FUNCTION_BLOCK FB_CapPreScrewer
VAR_INPUT
	bEnable								: BOOL;		//Zezwolenie na pracę
	bEstop								: BOOL;		//Stop awaryjny nieaktywny
	bHoming								: BOOL;		//Zezwolenie na wykonanie bazowania
	bIgnoreError						: BOOL;		//Ignorowania błędów cyklu pracy
	
	bReset								: BOOL;		//Reset błędu, jeśli w stanie "eError
	bManualMovement						: BOOL;		//Zezwolenie na ruchy ręcznę
	
	bRun								: BOOL;		//Rozkaz uruchomienia zakręcarki
	bPreRun								: BOOL;		//Przygotowanie stacji do pracy
	bSimulationEna						: BOOL;		//Tryb symulacji
	bPlacePermission					: BOOL;		//Zezwolenenie na wkładanie nakrentki w butelkę
	bMover1InPlacePos					: BOOL;		//Wózek 1 na pozycji Place
	bMover2InPlacePos					: BOOL;		//Wózek 2 na pozycji Place

	bCapSuckerVacumOk1					: BOOL;		//Sygnał podciśnienia na ssawce nakrętki 1
	bCapSuckerVacumOk2					: BOOL;		//Sygnał podciśnienia na ssawce nakrętki 2
	bCapSuckerVacumOk3					: BOOL;		//Sygnał podciśnienia na ssawce nakrętki 3
	bCapSuckerVacumOk4					: BOOL;		//Sygnał podciśnienia na ssawce nakrętki 4
	
	bStrawCatcherOut					: BOOL;		//Sygnał z krańcówki - wysunięty łapacz słomek
	bStrawCatcherIn						: BOOL;		//Sygnał z krańcówki - wysunięty łapacz słomek
	
	bStrawCatcherOpen1					: BOOL;		//Sygnał z krańcówki - otwart łapacz słomek 1
	bStrawCatcherOpen2					: BOOL;		//Sygnał z krańcówki - otwart łapacz słomek 2
	bStrawCatcherOpen3					: BOOL;		//Sygnał z krańcówki - otwart łapacz słomek 3
	bStrawCatcherOpen4					: BOOL;		//Sygnał z krańcówki - otwart łapacz słomek 4
	bSetEncoderOffsetAxisZ				: BOOL;		//Ustaw pozycję enkodera osi Z 
	
	stCommandsIn						: ST_CapPreScrewerCommandsIn;		

	stParameters						: ST_CapPreScrewerParameters;
	stMoverStatus						: ST_MoverState;
	
	iStationIndex						: UDINT;		//Numer stacji 
	wsStationName						: WSTRING;	//Nazwa stacji
	
END_VAR

VAR_OUTPUT
	eState							: E_Station;			//Stan ogólny bloku
	eRunningState					: E_CapPreScrewer; 		//Stan załapywarki
	bHomingDone						: BOOL;					//Stacja zbazowana
	bError							: BOOL;						//Błąd stacji
	udiErrorID						: UDINT;					//Nr błędu zakręcarki
	sErrorDescription				: STRING(200);				//Opis błędu
	sErrorDescription2				: STRING(200);				//Opis błędu
	sErrorStationName				: STRING;					//Nazwa stacj
	
	udiCartesianXServoErrorNr		: UDINT;					//Nr błędu serwa poziomego X
	udiCartesianZServoErrorNr		: UDINT;					//Nr błędu serwa pionowego Y
	udiPreScrewerServoErrorNr		: UDINT;					//Nr błędu serwa obrotowego załapywarki
	udiCatcherServoErrorNr			: UDINT;					//Nr błędu serwo pionowego uchwytu słomek
	
	_OUTPUT_						: BOOL;
	bBottleGrippers					: BOOL;						//Sygnał do zaworu - łapania szyjek butelek

	bCapSucker 						: ARRAY [1..4] OF BOOL;		//Sygnał do zaworu - zassij nakrętkę
	//bCapSucker2						: BOOL;						//Sygnał do zaworu - zassij nakrętkę 2
	//bCapSucker3						: BOOL;						//Sygnał do zaworu - zassij nakrętkę 3
	//bCapSucker4						: BOOL;						//Sygnał do zaworu - zassij nakrętkę 4
	
	bCapBlower1						: BOOL;						//Sygnał do zaworu - wydmuchaj nakrętkę 1
	bCapBlower2						: BOOL;						//Sygnał do zaworu - wydmuchaj nakrętkę 2
	bCapBlower3						: BOOL;						//Sygnał do zaworu - wydmuchaj nakrętkę 3
	bCapBlower4						: BOOL;						//Sygnał do zaworu - wydmuchaj nakrętkę 4
	
	bCapCatcher1					: BOOL;						//Sygnał do zaworu - złap nakrętkę 1
	bCapCatcher2					: BOOL;						//Sygnał do zaworu - złap nakrętkę 2
	bCapCatcher3					: BOOL;						//Sygnał do zaworu - złap nakrętkę 3
	bCapCatcher4					: BOOL;						//Sygnał do zaworu - złap nakrętkę 4
	
	bStrawCatchersOpen				: BOOL;						//Sygnał do zaworu - otwórz chwytaki słomek
	bStrawCatchersClose				: BOOL;						//Sygnał do zaworu - zamknij chwytaki słomek
	
	bStrawCatcherActuatorOut		: BOOL;						//Sygnał do zaworu - wysuń łapacz słomek
	bStrawCatcherActuatorIn			: BOOL;						//Sygnał do zaworu - wsuń łapacz słomek
	bMissingCaps					: BOOL;						//Żadna nakretka nie zostala pobrana
	
	bCycleDone						: BOOL;						//Cykl zakończono
	bCycleNotDone					: BOOL;						//Nie zakończono cyklu przestawiania wózków
	aCapPresence					: ARRAY [1..4] OF BOOL;		//jakie nakretki zostaly odlozone do butelek
	bAxisYSafePos					: BOOL;						//Bezpieczna pozycja osi Y dla przejazdu mówerów
	bCartesianSafePos				: BOOL;						//Bezpieczna pozycja kartezjana dla przejazdu mówerów
	bRejectDone						: BOOL;						// Zakończony odrzut
END_VAR

VAR_IN_OUT
	bStepButton						: BOOL; 		//Następny krok sekwencji	

	bManualBottleGripperUp			: BOOL;			//Ręczny ruch Jisang
	bManualBottleGripperDown		: BOOL;			//Ręczny ruch Jisang
	
	bManualCartesianYJogPlus		: BOOL;			//Ruch ręczny podajnika zamknięć 
	bManualCartesianYJogMinus		: BOOL;			//Ruch ręczny podajnika zamknięć 
	bManualCartesianZJogPlus		: BOOL;			//Ruch ręczny podajnika zamknięć 
	bManualCartesianZJogMinus		: BOOL;			//Ruch ręczny podajnika zamknięć 
	
	bManualPreScrewerJogPlus		: BOOL;
	bManualPreScrewerJogMinus		: BOOL;
	
	bManualCatcherJogPlus			: BOOL;
	bManualCatcherJogMinus			: BOOL;

	bManualCapSucker1				: BOOL;						//Ręczne sterowanie zaworu - zassij nakrętkę 1
	bmanualCapSucker2				: BOOL;						//Ręczne sterowanie - zassij nakrętkę 2
	bManualCapSucker3				: BOOL;						//Ręczne sterowanie - zassij nakrętkę 3
	bManualCapSucker4				: BOOL;						//Ręczne sterowanie - zassij nakrętkę 4
	                                
	bManualCapBlower1				: BOOL;						//Ręczne sterowanie - wydmuchaj nakrętkę 1
	bManualCapBlower2				: BOOL;						//Ręczne sterowanie - wydmuchaj nakrętkę 2
	bManualCapBlower3				: BOOL;						//Ręczne sterowanie - wydmuchaj nakrętkę 3
	bManualCapBlower4				: BOOL;						//Ręczne sterowanie - wydmuchaj nakrętkę 4
	
	bManualCapCatcher1				: BOOL;						//Ręczne sterowanie - złap nakrętkę 1
	bManualCapCatcher2				: BOOL;						//Ręczne sterowanie - złap nakrętkę 2
	bManualCapCatcher3				: BOOL;						//Ręczne sterowanie - złap nakrętkę 3
	bManualCapCatcher4				: BOOL;						//Ręczne sterowanie - złap nakrętkę 4
	
	bManualStrawCatchersOpen		: BOOL;						//Ręczne sterowanie - zamknij chwytaki słomek
	bManualStrawCatchersClose		: BOOL;                     //Ręczne sterowanie - otwórz chwytaki słomek
	                                  
	bManualStrawCatcherActuatorOut	: BOOL;						//Ręczne sterowanie - wysuń łapacz słomek
	bManualStrawCatcherActuatorIn	: BOOL;                     //Ręczne sterowanie - wsuń łapacz słomek
	
	CartesianYAxisRef				: AXIS_REF;		//Struktura sterowania NC dla serwa przesuwania poziomego
	CartesianZAxisRef				: AXIS_REF;		//Struktura sterowania NC dla serwa przesuwania pionowego
	PreScrewerAxisRef				: AXIS_REF;		//Struktura sterowania NC dla serwa załapywania nakrętek
	CatcherAxisRef					: AXIS_REF;		//Struktura sterowania NC dla serwa prowadzenia słomki
	bAdvancedHoming: BOOL;
END_VAR

VAR
	fbStrawCatcherLift				: FB_Checker;

	diMover1VacuumRetry				: ARRAY [1..4] OF DINT;					// Ilość prób pobrania wózek 1, słoty 1..4
	diMover2VacuumRetry				: ARRAY [1..4] OF DINT;					// Ilość prób pobrania wózek 2, słoty 1..4
	
	tonDelayServoOn					: TON;
	
	mcCartesianYManualMove			: MC_JOG; 			// Blok ruchu ręcznego 
	mcCartesianZManualMove			: MC_JOG; 			// Blok ruchu ręcznego
	mcPreScrewerManualMove			: MC_JOG; 			// Blok ruchu ręcznego
	mcCatcherManualMove				: MC_JOG; 			// Blok ruchu ręcznego
	
	mcCartesianYStop				: MC_Stop;			// Trwałe zatrzymywanie Serwo
	mcCartesianZStop				: MC_Stop;			// Trwałe zatrzymywanie Serwo
	mcPreScrewerStop				: MC_Stop;			// Trwałe zatrzymywanie Serwo
	mcCatcherStop					: MC_Stop;			// Trwałe zatrzymywanie Serwo
	
	mcCatcherHalt				: MC_Halt;			// Trwałe zatrzymywanie Serwo
	
//	mcMover1MoveVelocity		: MC_MoveVelocity;		// Ruch prędkościowy
//	mcMover2MoveVelocity		: MC_MoveVelocity;		// Ruch prędkościowy
//	mcMover1MoveVelocity2		: MC_MoveVelocity;		// Ruch prędkościowy
//	mcMover2MoveVelocity2		: MC_MoveVelocity;		// Ruch prędkościowy	
//	mcMover1MoveRelative		: MC_MoveRelative; 		// Ruch relatywny
	
	mcCartesianYMoveAbsolute	: MC_MoveAbsolute; 		// Ruch absolutny
	mcCartesianYMoveRelative	: MC_MoveRelative;		// Ruch względny
	mcCartesianZMoveAbsolute	: MC_MoveAbsolute; 		// Ruch absolutny
	mcCartesianZMoveAbsolute2	: MC_MoveAbsolute; 		// Ruch absolutny
	mcPreScrewerMoveAbsolute	: MC_MoveAbsolute; 		// Ruch absolutny
	mcPreScrewerMoveRelative	: MC_MoveRelative; 		// Ruch względny
	mcCatcherMoveAbsolute		: MC_MoveAbsolute; 		// Ruch absolutny
	
	fbAxisYPositioningOffset	: FB_CoEAX8000SetPositionOffset;
	fbAxisZPositioningOffset	: FB_CoEAX8000SetPositionOffset;
	
	mcCartesianYPower			: MC_Power;			 	// Zasilanie napędu
	mcCartesianZPower			: MC_Power;			 	// Zasilanie napędu
	mcPreScrewerPower			: MC_Power;			 	// Zasilanie napędu
	mcCatcherPower				: MC_Power;			 	// Zasilanie napędu
	
	mcPreScrewerHome			: MC_Home;	
	
	bCartesianYServoPower		: BOOL;					// Zmienna sterujaca zasilaniem serwo
	bCartesianZServoPower		: BOOL;					// Zmienna sterujaca zasilaniem serwo	
	bPreScrewerPower			: BOOL;					// Zmienna sterujaca zasilaniem serwo
	bCatcherPower				: BOOL;					// Zmienna sterujaca zasilaniem serwo
	
	fbCartesianYHardReset		: FB_SoEReset; 			// Blok twardego resetu serwa
	fbCartesianZHardReset		: FB_SoEReset; 			// Blok twardego resetu serwa
	fbPreScrewerHardReset		: FB_SoEReset; 			// Blok twardego resetu serwa
	fbCatcherHardReset			: FB_SoEReset; 			// Blok twardego resetu serwa
	mcCartesianYSoftReset		: MC_Reset; 			// blok łagodnego resetu serwa 
	mcCartesianZSoftReset		: MC_Reset; 			// blok łagodnego resetu serwa
	mcPreScrewerSoftReset		: MC_Reset; 			// blok łagodnego resetu serwa
	mcCatcherSoftReset			: MC_Reset; 			// blok łagodnego resetu serwa
	
	(*Bledy, Resetowanie*)
	tonResetting						: TON;
	rtResetCommands						: R_TRIG;
	tonActualMotor1TemperatureTooHigh	: TON;
	tonActualMotor2TemperatureTooHigh	: TON;
		
	bStateError							: BOOL;
	
	eLastState					: E_Station;			// Stan ogólny bloku
	eLastRunningState			: E_CapPreScrewer;		// Stan podbloku
	eLastStateTemp				: E_Station;			// Stan ogólny bloku
	//eLastRunningStateTemp		: E_CapFeeder;		// Stan podbloku
	
	(*Casy od różnych stanów*)
	iAbortingCASE				: INT;
	iStoppingCase 				: INT;
	iHomingCase					: INT;
	iErrorResseting2			: INT;
	iTestResetting				: INT;
	iCountAborting				: INT;
	
	(*Filtry czujników*)
	tonSuckedOk					: ARRAY [1..4] OF TON;
	//tonSuckedOk2				: TON;
	//tonSuckedOk3				: TON;
	//tonSuckedOk4				: TON;
	
	tonStrawCatcherIn			: TON;
	tonStrawCatcherOut			: TON;
	
	tonStrawCatcher1Open		: TON;
	tonStrawCatcher2Open		: TON;
	tonStrawCatcher3Open		: TON;
	tonStrawCatcher4Open		: TON;
	
	tonStrawCatcher1Close		: TON;
	tonStrawCatcher2Close		: TON;
	tonStrawCatcher3Close		: TON;
	tonStrawCatcher4Close		: TON;
	
	//Czasówki do obsługi błędów siłowników
	tonErrorStrawCatcherIn		: TON;
	tonErrorStrawCatcherOut		: TON;
	
	tonErrorStrawCatcherOpen1	: TON;
	tonErrorStrawCatcherOpen2	: TON;
	tonErrorStrawCatcherOpen3	: TON;
	tonErrorStrawCatcherOpen4	: TON;
	
	//Czasówki do obsługi problemu z zasysaniem
	tonErrorSuckerVacum1		: TON;
	tonErrorSuckerVacum2		: TON;
	tonErrorSuckerVacum3		: TON;
	tonErrorSuckerVacum4		: TON;
	tonCapCatcher				: TON;
	
	tonBlowOFF					: TON;
	bCapsBlowON					: BOOL;
	
	tonVacuumWatchdog			: TON;
	i: INT;
	
	tonBlowerON				: ARRAY [1..4] OF TON;	//Cap blowing timers
		
	tonPlacePermission			: TON;
	rtPlacePermission			: R_TRIG;
	bGripperOpen: BOOL;
	bStopAllowed: BOOL;
	
//	fbBottleCatch									: fb
	eBottleCatch1State								:E_Station; 						// Stan chwytaka stabilizujšcego pod podajnikiem nakrętek
	eBottleCatch2State								:E_Station; 						// Stan chwytaka stabilizujšcego pod podajnikiem nakrętek
	eBottleCatch3State								:E_Station; 						// Stan chwytaka stabilizujšcego pod podajnikiem nakrętek
	eBottleCatch4State								:E_Station; 						// Stan chwytaka stabilizujšcego pod podajnikiem nakrętek
	eBottleCatch1RunningState						:E_CatchStationState; 				// Poprzedni stan chwytaka pod podajnikiem nakrętek
	eBottleCatch2RunningState						:E_CatchStationState; 				// Poprzedni stan chwytaka pod podajnikiem nakrętek
	eBottleCatch3RunningState						:E_CatchStationState; 				// Poprzedni stan chwytaka pod podajnikiem nakrętek
	eBottleCatch4RunningState						:E_CatchStationState; 				// Poprzedni stan chwytaka pod podajnikiem nakręte
	fbBottleCatch1State								:FB_State;
	fbBottleCatch2State								:FB_State;
	fbBottleCatch3State								:FB_State;
	fbBottleCatch4State								:FB_State;
	
	IbBottleCatchHeightMotorEncoderPulse			: BOOL;									// Sygnał impulsów enkodera siłownika	
                                            
                                                    
    QbBottleCatchHeightUpCmd              			: BOOL;  								// Zmienna sterownika bezpośrednio sterująca siłownikiem w górę 
    QbBottleCatchHeightDownCmd            			: BOOL;									// Zmienna sterownika bezpośrednio sterująca siłownikiem w dół 	
	bBottleCatcherCatchTemp							: BOOL;
	rtRun											: R_TRIG;
	bTestStrawCatcher								: BOOL;
	bTestError										: BOOL;
	bCatcHActuator1									: BOOL;
	bCatcHActuator2									: BOOL;
	bCatcHActuator3									: BOOL;
	bCatcHActuator4									: BOOL;
                                                	
	bCollisionWithMoverArea							: BOOL;
	bCollisionError									: BOOL;
	bCollision1Error								: BOOL;
	bCollision2Error								: BOOL;
	rtCollisionError								: R_TRIG;
	tonCollisionError								: TON;
	bCapBlow1										: BOOL;
	bCapBlow2										: BOOL;
	bCapBlow3										: BOOL;
	bCapBlow4										: BOOL;
	bPlaceDone										: BOOL;
	bTestCatch										: BOOL;
	iDisablingCase									: INT;
	bAdditionalBlow									: BOOL;
	bAxisYInPosition								: BOOL;
	bAxisZInPosition								: BOOL;
	bAxisZInPosition1								: BOOL;
	bAxisZInPosition2								: BOOL;
	bHomingWithoutJiesang							: BOOL;
	bCapLost										: ARRAY [1..4] OF BOOL;
	bAnyCapLost										: BOOL;

	trStepButton: R_TRIG;
	diManualModeCase								: DINT;
	bAxisYInHomePos									: BOOL;
	bAxisZInHomePos									: BOOL;
	bAxisZInTopPos									: BOOL;
	bAxisStrawCatcherHomePos						: BOOL;
	bCartesianInHomePos								: BOOL;										//Kartezjan znajduje sie na poz. home
	bCartesianInTopPos								: BOOL;
	bCartesianReady									: BOOL;										//Kartezjan gotowy do sekwencji
	rtCheckVacuumPart4								: R_TRIG;	


	FB_AxisY_ADS_Read								: FB_EcCoESdoRead;
	uiAxisY_ADS_Read								: UINT;
	tonAxisY_ADS_Read							    : TON;
	
	stAxisY_ADS										: ST_ADS_Read_Write;
	iAxisY_ADS_ReadCase								: INT;
	
	ftAxisY_ADS_Read								: F_TRIG;
	
	ftAxisY_ADS_Write								: F_TRIG;
	
	bSetPosition									: BOOL;
	FB_AxisY_ADS_Write								: FB_EcCoESdoWrite;
	tonAxisYLagDetction								: TON;		
	bCartesianInReadyPos							: BOOL;
	lrPreScrewerAxisSavedPosition					: LREAL;
	lrAxisZSavedPosition							: LREAL;
	
	bChangeSpeedRightLeft							: BOOL;
	rtPendantRightLeftFast							: R_TRIG;
	ftPendantRightLeftFast							: F_TRIG;
	bChangeSpeedUpDown								: BOOL;
	rtPendantUpDownFast								: R_TRIG;
	ftPendantUpDownFast								: F_TRIG;
	
	bAnyCapPresence									: BOOL;		//Obecna przynajmniej jedna nasadka
	tonWaitInPlacePos								: TON;
	diPreSCrewerHomePos								: DINT;

	//Synchronizacja osi podczas prowadzenia slomki
	fbGearInAxisZ									: MC_GearInDyn;
	fbGearInAxisZ_Screwer							: MC_GearIn;	
	fbGearInCatcherAxis								: MC_GearInDyn;
	fbGearOutAxisZ									: MC_GearOut;
	fbGearOutCatcherAxis							: MC_GearOut;
	fbVirtualAxis									: FB_AxisAX8000;
	fbGearInPos										: MC_GearInPos; 
	VirtualEna										: BOOL := TRUE;
	
	fbCamTableSelectAxisZ							: MC_CamTableSelect;
	fbCamInAxisZ									: MC_CamIn;
	fbCamOutAxisZ									: MC_CamOut;
	fbCamTableSelectCatcher							: MC_CamTableSelect;
	fbCamInAxisCatcher								: MC_CamIn;
	fbCamOutAxisCatcher								: MC_CamOut;	
	
	stCamTableIdAxisZ								: MC_CAM_ID;
	stCamTableAxisZRef								: MC_CAM_REF;
	arrTableAxisZ									: ARRAY[0..2, 0..1] OF LREAL;
	stCamTableIdCatcher								: MC_CAM_ID;
	stCamTableCatcherRef							: MC_CAM_REF;
	arrTableCatcher									: ARRAY[0..2, 0..1] OF LREAL;
	
	nAxisYSafetyState			AT%I*				: BYTE;	//Satatus safety 
	nAxisZSafetyState			AT%I*				: BYTE;	//Satatus safety 
	nAxisScrewSafetyState		AT%I*				: BYTE;	//Satatus safety 
	nAxisCatcherSafetyState		AT%I*				: BYTE;	//Satatus safety 
	
	uiAxisYTorqueLimit			AT%Q*				: UINT;
	
	rtChoseRecipe									: R_TRIG;
	tonCapCatcher1Open								: TON;
	bVirtualMove									: BOOL;		//Absolutny ruch  wirtualnej osi
	rtMove											: R_TRIG;
	ftMove											: F_TRIG;
	bVirtualAxisMove1								: BOOL;		//Ruch 1 wirtualnej osi
	bVirtualAxisMove2								: BOOL;		//Ruch 2 wirtualnej osi
	
	nMoveId											: INT;		//
	stVirtualMove_Out								: Tc2_MC2.ST_McOutputs;
	stVirtualMove1_Out								: Tc2_MC2.ST_McOutputs;	//struktura wyjsciowa ruchu wirtualnej osi
	stVirtualMove2_Out								: Tc2_MC2.ST_McOutputs; //struktura wyjsciowa ruchu wirtualnej osi
	bEnableLift										: BOOL	:= TRUE;
	bStrawCatcherLiftInHomePos						: BOOL;
	bMover1InPickPos								: BOOL; 			//nakrętka pobrana z wózka nr1
	bCapScrewed										: BOOL;				// nakrętka zakręcona
	rtSetEncoderOffsetAxisZ							: R_TRIG;
	tonStrawCatcherLiftInHomePos					: TON;				//łapacz słomek jest na poz bazowej
//	lrCatcherOffsetRegardingAxisZ					: LREAL;			//różnica położenia łapacza słomek odnośnie osi Z		
	bAlarmInit										: BOOL := TRUE;
	arrFbAllarm										: ARRAY [0..29] OF FB_TcAlarm;
	fbSourceInfo 									: FB_TcSourceInfo;
	sAxisAlarm										: STRING;	
	iSimulationCase									: INT;		
	bStrawCatcherLiftEnable							: BOOL;
	bReject											: BOOL;			//Odrzut aktywowany
	bTubeReject										: BOOL;			//Odrzut poprzez brak słomki
	iRejectCase										: INT;			
	lrAxisZ_RejectOffset							: LREAL;		//Offset odrzutu
	bAllSlotsVacuumStatus							: BOOL;			//Status wszsystkich aktywowanych ssawek
	arrVacuumStatus									: ARRAY [1..4] OF BOOL;	//status pojedynczych gniazd
	rtAxisZMoving									: R_TRIG;
	
	bTestCamCalculation								: BOOL;
END_VAR

IF bAlarmInit THEN
	ACT_ErrorInit();
END_IF


GVL_VIS.lrCapSorterPreScrewerStrawCatcherCVShow 			:= CatcherAxisRef.NcToPlc.ActPos;
GVL_VIS.lrCapSorterPreScrewerYAxisCVShow					:= CartesianYAxisRef.NcToPlc.ActPos;
GVL_VIS.lrCapSorterPreScrewerZAxisCVShow					:= CartesianZAxisRef.NcToPlc.ActPos;
GVL_VIS.lrCapSorterPreScrewerCAxisCVShow					:= PreScrewerAxisRef.NcToPlc.ActPos;

Signals();
ADS_Control();
Control();
ErrorHandling();
FBs();
CollisionAvoidance();


IF VirtualEna THEN
	ACT_VirtualAxisControl();
ELSE
	IF fbVirtualAxis.bEnable THEN
		fbVirtualAxis.Disable();
	END_IF	
END_IF

IF bTestCamCalculation THEN
	CamCalculation();
END_IF

ACTION ACT_ErrorInit:
bAlarmInit			:= FALSE;
fbSourceInfo.Clear();
fbSourceInfo.sName	:= wsLiteral_TO_UTF8(wsStationName);
fbSourceInfo.nId	:= iStationIndex;

arrFbAllarm[0].CreateEx(stEventEntry := TC_EVENTS.AlarmClass.CapPreScrewer_1130	, bWithConfirmation := FALSE, ipSourceInfo := fbSourceInfo);
arrFbAllarm[1].CreateEx(stEventEntry := TC_EVENTS.AlarmClass.CapPreScrewer_1131, bWithConfirmation := FALSE, ipSourceInfo := fbSourceInfo);
arrFbAllarm[2].CreateEx(stEventEntry := TC_EVENTS.AlarmClass.CapPreScrewer_1132, bWithConfirmation := FALSE, ipSourceInfo := fbSourceInfo);
arrFbAllarm[3].CreateEx(stEventEntry := TC_EVENTS.AlarmClass.CapPreScrewer_1133, bWithConfirmation := FALSE, ipSourceInfo := fbSourceInfo);
arrFbAllarm[4].CreateEx(stEventEntry := TC_EVENTS.AlarmClass.CapPreScrewer_1134, bWithConfirmation := FALSE, ipSourceInfo := fbSourceInfo);
arrFbAllarm[5].CreateEx(stEventEntry := TC_EVENTS.AlarmClass.CapPreScrewer_1135, bWithConfirmation := FALSE, ipSourceInfo := fbSourceInfo);
arrFbAllarm[6].CreateEx(stEventEntry := TC_EVENTS.AlarmClass.CapPreScrewer_1136, bWithConfirmation := FALSE, ipSourceInfo := fbSourceInfo);
arrFbAllarm[7].CreateEx(stEventEntry := TC_EVENTS.AlarmClass.CapPreScrewer_1137, bWithConfirmation := FALSE, ipSourceInfo := fbSourceInfo);
arrFbAllarm[8].CreateEx(stEventEntry := TC_EVENTS.AlarmClass.CapPreScrewer_1138, bWithConfirmation := FALSE, ipSourceInfo := fbSourceInfo);
arrFbAllarm[9].CreateEx(stEventEntry := TC_EVENTS.AlarmClass.CapPreScrewer_1139, bWithConfirmation := FALSE, ipSourceInfo := fbSourceInfo);
arrFbAllarm[10].CreateEx(stEventEntry := TC_EVENTS.AlarmClass.CapPreScrewer_1140, bWithConfirmation := FALSE, ipSourceInfo := fbSourceInfo);
arrFbAllarm[11].CreateEx(stEventEntry := TC_EVENTS.AlarmClass.CapPreScrewer_1141, bWithConfirmation := FALSE, ipSourceInfo := fbSourceInfo);
arrFbAllarm[12].CreateEx(stEventEntry := TC_EVENTS.AlarmClass.CapPreScrewer_1142, bWithConfirmation := FALSE, ipSourceInfo := fbSourceInfo);
arrFbAllarm[13].CreateEx(stEventEntry := TC_EVENTS.AlarmClass.CapPreScrewer_1143, bWithConfirmation := FALSE, ipSourceInfo := fbSourceInfo);
arrFbAllarm[14].CreateEx(stEventEntry := TC_EVENTS.AlarmClass.CapPreScrewer_1144, bWithConfirmation := FALSE, ipSourceInfo := fbSourceInfo);
arrFbAllarm[15].CreateEx(stEventEntry := TC_EVENTS.AlarmClass.CapPreScrewer_1145, bWithConfirmation := FALSE, ipSourceInfo := fbSourceInfo);
arrFbAllarm[16].CreateEx(stEventEntry := TC_EVENTS.AlarmClass.CapPreScrewer_1146, bWithConfirmation := FALSE, ipSourceInfo := fbSourceInfo);
arrFbAllarm[17].CreateEx(stEventEntry := TC_EVENTS.AlarmClass.CapPreScrewer_1147, bWithConfirmation := FALSE, ipSourceInfo := fbSourceInfo);
arrFbAllarm[18].CreateEx(stEventEntry := TC_EVENTS.AlarmClass.CapPreScrewer_1148, bWithConfirmation := FALSE, ipSourceInfo := fbSourceInfo);
arrFbAllarm[19].CreateEx(stEventEntry := TC_EVENTS.AlarmClass.CapPreScrewer_1149, bWithConfirmation := FALSE, ipSourceInfo := fbSourceInfo);
arrFbAllarm[20].CreateEx(stEventEntry := TC_EVENTS.AlarmClass.CapPreScrewer_1150, bWithConfirmation := FALSE, ipSourceInfo := fbSourceInfo);
arrFbAllarm[21].CreateEx(stEventEntry := TC_EVENTS.AlarmClass.CapPreScrewer_1151, bWithConfirmation := FALSE, ipSourceInfo := fbSourceInfo);
arrFbAllarm[22].CreateEx(stEventEntry := TC_EVENTS.AlarmClass.CapPreScrewer_1152, bWithConfirmation := FALSE, ipSourceInfo := fbSourceInfo);
arrFbAllarm[23].CreateEx(stEventEntry := TC_EVENTS.AlarmClass.CapPreScrewer_1153, bWithConfirmation := FALSE, ipSourceInfo := fbSourceInfo);
arrFbAllarm[24].CreateEx(stEventEntry := TC_EVENTS.AlarmClass.CapPreScrewer_1154, bWithConfirmation := FALSE, ipSourceInfo := fbSourceInfo);
arrFbAllarm[25].CreateEx(stEventEntry := TC_EVENTS.AlarmClass.CapPreScrewer_1155, bWithConfirmation := FALSE, ipSourceInfo := fbSourceInfo);
arrFbAllarm[26].CreateEx(stEventEntry := TC_EVENTS.AlarmClass.CapPreScrewer_1156, bWithConfirmation := FALSE, ipSourceInfo := fbSourceInfo);
arrFbAllarm[27].CreateEx(stEventEntry := TC_EVENTS.AlarmClass.CapPreScrewer_1157, bWithConfirmation := FALSE, ipSourceInfo := fbSourceInfo);
arrFbAllarm[28].CreateEx(stEventEntry := TC_EVENTS.AlarmClass.CapPreScrewer_1158, bWithConfirmation := FALSE, ipSourceInfo := fbSourceInfo);
arrFbAllarm[29].CreateEx(stEventEntry := TC_EVENTS.AlarmClass.CapPreScrewer_1159, bWithConfirmation := FALSE, ipSourceInfo := fbSourceInfo);
END_ACTION

ACTION ACT_VirtualAxisControl:
IF fbVirtualAxis.bDisabled THEN
	fbVirtualAxis.bEnable	:= TRUE;
	fbVirtualAxis.Power();
END_IF


rtMove(CLK := bVirtualMove);
ftMove(CLK := bVirtualMove);

IF rtMove.Q THEN
	bVirtualAxisMove2 							S= stVirtualMove1_Out.Busy; 
	bVirtualAxisMove1 							S= NOT bVirtualAxisMove2;
ELSIF ftMove.Q THEN
	bVirtualAxisMove1							R= TRUE;	
    bVirtualAxisMove2							R= TRUE;	
END_IF


IF NOT stVirtualMove2_Out.Busy AND NOT stVirtualMove2_Out.Done THEN
	nMoveId					:= 1;
	stVirtualMove_Out		:= stVirtualMove1_Out ;
ELSE
	nMoveId					:= 2;
	stVirtualMove_Out		:= stVirtualMove2_Out;
END_IF

stVirtualMove1_Out 			:= fbVirtualAxis.MoveAbsolute(bExecute := bVirtualAxisMove1);
stVirtualMove2_Out 			:= fbVirtualAxis.MoveAbsolute2(bExecute := bVirtualAxisMove2);


fbVirtualAxis.fAcceleration;//						:= stParameters.lrPickerAcceleration;	//100_000_000.0;
fbVirtualAxis.fDeceleration;//						:= stParameters.lrPickerAcceleration;	//100_000_000.0;
fbVirtualAxis.fJerk;//							:= stParameters.lrPickerJerk;// 	1_000_000;//100_000_000_000;  








fbGearInPos.SyncMode.GearInSyncMode							:= E_GearInSyncMode.GEARINSYNCMODE_POSITIONBASED;	//Synchronizacja według pozycji mastera
fbGearInPos.SyncMode.GearInSync_OpMask_DetailedErrorCodes 	:= TRUE;	//szczególowy opis błedów
fbGearInPos.SyncMode.GearInSync_CheckMask_MaxVelo 			:= TRUE;	//vSlave | ≤ vSlaveMax
fbGearInPos.SyncMode.GearInSync_CheckMask_MaxAcc 			:= TRUE;	//accSlave ≤ accSlaveMax
fbGearInPos.SyncMode.GearInSync_CheckMask_MaxDec 			:= TRUE;	//decSlave ≤ decSlaveMax
fbGearInPos.SyncMode.GearInSync_CheckMask_MaxJerk 			:= TRUE;	//jSlave ≤ jSlaveMax
fbGearInPos.SyncMode.GearInSync_CheckMask_MinPos			:= TRUE;
fbGearInPos.SyncMode.GearInSync_CheckMask_MaxPos			:= TRUE;
fbGearInPos.Options.PositionLimitMax;//						:= 450.0;//SEL(stParameters.lrCartesianCatchZPosition>450, stParameters.lrCartesianCatchZPosition, 450);
fbGearInPos.Options.PositionLimitMin						:= 0.0;
END_ACTION

ACTION ADS_Control:
tonAxisY_ADS_Read(PT := T#250MS);

(*	//Wyłączenie krańcówek podczas bazowania na zderzak wózek 1
			IF eState = E_Station.eHoming AND bAdvancedHoming AND uiMover1ADS_Read <> 0 THEN	//	ADS_Read = 0 - no limit switch
				uiMover1ADS_Write				:= 0;                                           //			 = 1 - NC
				FB_Mover1ADS_Write.bExecute		:= TRUE;                                        //			 = 2 - NO
			ELSIF eState <> E_Station.eHoming AND uiMover1ADS_Read <> 1 THEN	                
				uiMover1ADS_Write				:= 1;                                           
				FB_Mover1ADS_Write.bExecute		:= TRUE;                                        
			END_IF
		
			ftMover1ADS_Write(CLK := FB_Mover1ADS_Write.bBusy);
			FB_Mover1ADS_Write.bExecute			R= ftMover1ADS_Write.Q;
			
		
	//Wyłączenie krańcówek podczas bazowania na zderzak wózek 2
			IF eState = E_Station.eHoming AND bAdvancedHoming AND uiMover2ADS_Read <> 0 THEN
				uiMover2ADS_Write				:= 0;
				FB_Mover2ADS_Write.bExecute		:= TRUE;
			ELSIF eState <> E_Station.eHoming AND uiMover2ADS_Read <> 1 THEN	 
				uiMover2ADS_Write				:= 1;
				FB_Mover2ADS_Write.bExecute		:= TRUE;
			END_IF
		\
			ftMover2ADS_Write(CLK := FB_Mover2ADS_Write.bBusy);
			FB_Mover2ADS_Write.bExecute			R= ftMover2ADS_Write.Q;
		
		
	//odswieżanie parametrów krańcówek hardwerowych wózek 1
			ftMover1ADS_Read(CLK := FB_Mover1ADS_Read.bBusy);
			FB_Mover1ADS_Read.bExecute			S= (tonAxisY_ADS_Read.Q AND NOT ftMover1ADS_Read.Q);
			FB_Mover1ADS_Read.bExecute			R= ftMover1ADS_Read.Q;
			
			tonAxisY_ADS_Read.IN				:= NOT tonAxisY_ADS_Read.Q;
	
	//odswieżanie parametrów krańcówek hardwerowych wózek 2
			ftMover2ADS_Read(CLK := FB_Mover2ADS_Read.bBusy);
			FB_Mover2ADS_Read.bExecute			S= (tonAxisZ_ADS_Read.Q AND NOT ftMover2ADS_Read.Q);
			FB_Mover2ADS_Read.bExecute			R= ftMover2ADS_Read.Q;
			
			tonAxisZ_ADS_Read.IN				:= NOT tonAxisZ_ADS_Read.Q;*)

////////////////////////////////////////////////////////////////////////////////////////////////////////////////

//CASE iAxisY_ADS_ReadCase OF
//	
//	0://Odczyt momentu
//	FB_AxisY_ADS_Read.nSubIndex				:= 16#0;
//	FB_AxisY_ADS_Read.nIndex				:= 16#60E0;
//	                                		
//	stAxisY_ADS.stSts.uiTorq				:= uiAxisY_ADS_Read;
//	                                		
//		IF ftAxisY_ADS_Read.Q THEN  		
//			iAxisY_ADS_ReadCase				:= 1;
//		END_IF
//	
//	1://Odczyt krancowek

//	
//END_CASE

		//Wyłączenie krańcówek podczas bazowania na zderzak oś Y
	IF eState = E_Station.eHoming AND bAdvancedHoming AND stAxisY_ADS.uiHardwerLimitSwitch <> 0 THEN//	ADS_Read = 0 - no limit switch
		FB_AxisY_ADS_Write.nSubIndex			:= 16#1;											//			 = 1 - NC
		FB_AxisY_ADS_Write.nIndex				:= 16#3003;                                         //			 = 2 - NO
		stAxisY_ADS.stCtr.siHardwerLimitSwitch	:= 0;                   
		FB_AxisY_ADS_Write.bExecute				:= TRUE;                
	ELSIF eState <> E_Station.eHoming AND stAxisY_ADS.uiHardwerLimitSwitch <> 1 THEN	
		FB_AxisY_ADS_Write.nSubIndex			:= 16#1;	
        FB_AxisY_ADS_Write.nIndex				:= 16#3003;
        stAxisY_ADS.stCtr.siHardwerLimitSwitch	:= 1;      
        FB_AxisY_ADS_Write.bExecute				:= TRUE;                                    
	END_IF
	
	ftAxisY_ADS_Write(CLK := FB_AxisY_ADS_Write.bBusy);
	FB_AxisY_ADS_Write.bExecute			R= ftAxisY_ADS_Write.Q;
	
	

	//odswieżanie parametrów krańcówek hardwerowych oś Y
	FB_AxisY_ADS_Read.nSubIndex					:= 16#1;
	FB_AxisY_ADS_Read.nIndex					:= 16#3003;
	
	ftAxisY_ADS_Read(CLK := FB_AxisY_ADS_Read.bBusy);
	FB_AxisY_ADS_Read.bExecute					S= (tonAxisY_ADS_Read.Q AND NOT ftAxisY_ADS_Read.Q);
	FB_AxisY_ADS_Read.bExecute					R= ftAxisY_ADS_Read.Q;
	stAxisY_ADS.uiHardwerLimitSwitch			:= uiAxisY_ADS_Read;
	
	tonAxisY_ADS_Read.IN						:= NOT tonAxisY_ADS_Read.Q;
	
	IF NOT bAdvancedHoming AND (stAxisY_ADS.stCtr.uiNegativeTorqueLimit <> 2000 OR stAxisY_ADS.stCtr.uiPositiveTorqueLimit <> 2000 OR uiAxisYTorqueLimit <> 2000) THEN	
		stAxisY_ADS.stCtr.uiNegativeTorqueLimit			:= 2000;	
		stAxisY_ADS.stCtr.uiPositiveTorqueLimit			:= 2000;
		uiAxisYTorqueLimit								:= 2000;
	END_IF
END_ACTION

ACTION CamCalculation:

//Tablica punktów dla osi prowadzenia słomki:
		//Pozycję Mastera:
	arrTableCatcher[0,0]			:= 0.0;		//Początek ruchu 
	arrTableCatcher[1,0]			:= (stParameters.lrCatcherCatchingPosition  - (stParameters.lrBottleHight - stParameters.lrCatcherHightSV - 40));	//Punkt nad butelką 40mm ---> 40mm grubość chwytaków /////
	//Sprawdzanie czy nie przekraczamy dolny limit (min 2mm)
	arrTableCatcher[1,0]			:= SEL((stParameters.lrCatcherCatchingPosition - arrTableCatcher[1,0] < 2.0), arrTableCatcher[1,0], (stParameters.lrCatcherCatchingPosition - 2.0));
	arrTableCatcher[2,0]			:= 1000.0;	//Koniec dojazdu mastera
	                        		
		//Pozycję Slave:    		
	arrTableCatcher[0,1]			:= 0.0;	//Początek ruchu 
	arrTableCatcher[1,1]			:= arrTableCatcher[1,0];	//Punkt nad butelką
	arrTableCatcher[2,1]			:= arrTableCatcher[1,0];	//Koniec dojazdu mastera

//Tablica punktów dla osi Z:
		//Pozycję Mastera:
	arrTableAxisZ[0,0]				:= 0.0;	//Początek ruchu 
	arrTableAxisZ[1,0]				:= (stParameters.lrCapHight - GVL_Recipe.lrCapSorterCapNeckHightShow - GVL_Recipe.lrCapSorterPreScrewerCheckValveShow - 30.0);	//Punkt Synchronizacji (~10mm od końca słomki)
	arrTableAxisZ[2,0]				:= 1000.0;	//Koniec dojazdu mastera
		//Pozycję Slave:    		
	arrTableAxisZ[0,1]				:= 0.0;	//Początek ruchu 
	arrTableAxisZ[1,1]				:= 0.0;	//Punkt Synchronizacji (~10mm od końca słomki)
	arrTableAxisZ[2,1]				:= 1000.0 - arrTableAxisZ[1,0];	//Koniec dojazdu mastera

//stCamTableCatcherRef.pArray			:= ADR(arrTableCatcher);
//stCamTableCatcherRef.ArraySize		:= SIZEOF(arrTableCatcher);
//stCamTableCatcherRef.TableType		:= MC_TableType.MC_TABLETYPE_NONEQUIDISTANT;
//stCamTableCatcherRef.NoOfRows		:= 3;
//stCamTableCatcherRef.NoOfColumns 	:= 2;
//stCamTableIdCatcher					:= SEL(stCamTableIdCatcher=0, stCamTableIdCatcher, 1);
//
//stCamTableAxisZRef.pArray			:= ADR(arrTableAxisZ);
//stCamTableAxisZRef.ArraySize		:= SIZEOF(arrTableAxisZ);
//stCamTableAxisZRef.TableType		:= MC_TableType.MC_TABLETYPE_NONEQUIDISTANT;
//stCamTableAxisZRef.NoOfRows			:= 3;
//stCamTableAxisZRef.NoOfColumns 		:= 2;
//stCamTableIdAxisZ					:= SEL(stCamTableIdAxisZ=0, stCamTableIdAxisZ, 2);
END_ACTION

ACTION CollisionAvoidance:

//bCollision1Error			:= 	mcCartesianYPower.Override = 0;
//bCollision2Error			:= 	mcCartesianZPower.Override = 0 OR mcCartesianZStop.Execute = TRUE;

tonCollisionError(IN := bCollision1Error OR bCollision1Error, PT := T#3S);
rtCollisionError(CLK := tonCollisionError.Q);

bCollisionWithMoverArea := CartesianZAxisRef.NcToPlc.ActPos < 354.0 AND CartesianYAxisRef.NcToPlc.ActPos < 65.0;

IF CartesianZAxisRef.NcToPlc.ActPos < 206 AND NOT bSetPosition THEN	
	
	IF CartesianYAxisRef.NcToPlc.SetPos <= 354 AND NOT CartesianYAxisRef.Status.PositiveDirection THEN
		mcCartesianYPower.Override 	:= 0;
//		bHomingDone					:= FALSE;
//	ELSIF CartesianYAxisRef.NcToPlc.SetPos >= 111 AND NOT CartesianYAxisRef.Status.NegativeDirection THEN
//		mcCartesianYPower.Override 	:= 0;
	ELSIF CartesianYAxisRef.Status.PositiveDirection THEN
		mcCartesianYPower.Override 	:= 100;	
	END_IF	
	
ELSE
	mcCartesianYPower.Override := 100;	
END_IF


//IF CartesianYAxisRef.NcToPlc.ActPos < 160 AND CartesianZAxisRef.NcToPlc.SetPos < 358 
//	OR CartesianYAxisRef.NcToPlc.ActPos > 200 AND CartesianZAxisRef.NcToPlc.SetPos < 185 THEN
//	
//		IF CartesianZAxisRef.Status.NegativeDirection AND CartesianZAxisRef.Status.Moving THEN
//			mcCartesianZStop.Execute						:= TRUE;
//			mcCartesianZMoveAbsolute.Execute				:= FALSE;
//			mcCartesianZMoveAbsolute2.Execute				:= FALSE;
//			
//			bHomingDone					:= FALSE;
//		ELSE
//			mcCartesianZStop.Execute						:= FALSE;
//		END_IF
//END_IF


//IF CartesianYAxisRef.NcToPlc.ActPos > 200 AND CartesianZAxisRef.NcToPlc.ActPos - CatcherAxisRef.NcToPlc.ActPos < 200 THEN
//	mcCartesianZPower.Override :=F_Scaling_Limit(
//									In:=ABS(CartesianZAxisRef.NcToPlc.ActPos - CatcherAxisRef.NcToPlc.ActPos),
//									INMin:=0, INMax:= 200, OUTMin:=0, OUTMax:=100);
//ELSE
//	mcCartesianZPower.Override	:= 100;
//END_IF



CartesianZAxisRef.NcToPlc.ActPos;
CartesianZAxisRef.PlcToNc.ExtSetPos;

CartesianYAxisRef.NcToPlc.ActPos;
CartesianYAxisRef.PlcToNc.ExtSetPos;
END_ACTION

ACTION Control:
	(** TIMERY**)
//	tonGripper1ReliseDelay	(IN:=	NOT bGripper1Actuator, 					PT:=T#50MS);	//bylo 80
//	tonGripper2ReliseDelay	(IN:=	NOT bGripper2Actuator, 					PT:=T#50MS);	//bylo 80
                                 	
//	tonGripper1Delay		(IN:=	bGripper1Actuator OR iTool = 2, 						PT:=T#150MS);	//bylo 200  /// jednak 150
//	tonGripper2Delay		(IN:=	bGripper2Actuator OR iTool = 2, 						PT:=T#150MS);	//bylo 200 /// a jednak 150
                            																																								// Nie moze być 60 bo nalicza 60 i powyzej 360 sie przekręca																			
//	tonTightScrewing1Timer	(IN:=	(eRunningState=E_GripperScrewer.eScrewing) AND NOT tonTightScrewing1Timer.Q AND mcScrewer1MoveVelocity.Execute AND mcScrewer1MoveVelocity.InVelocity AND Screwing1AxisRef.NcToPlc.ActVelo < 100 (*AND ABS(Screwing1AxisRef.NcToPlc.PosDiff)>60 *) AND NOT bScrewed1,PT:=INT_TO_TIME(iScrewTightTime));
//	tonTightScrewing2Timer	(IN:=	(eRunningState=E_GripperScrewer.eScrewing) AND NOT tonTightScrewing2Timer.Q AND mcScrewer2MoveVelocity.Execute AND mcScrewer2MoveVelocity.InVelocity AND Screwing2AxisRef.NcToPlc.ActVelo < 100 (*AND ABS(Screwing2AxisRef.NcToPlc.PosDiff)>60 *) AND NOT bScrewed2,PT:=INT_TO_TIME(iScrewTightTime));

//	tonTightScrewing1TimerAndOpenedGripper(IN:=bScrewed1,	PT:=T#100MS);
//	tonTightScrewing2TimerAndOpenedGripper(IN:=bScrewed2,	PT:=T#100MS);	
	
//	tonMomentaryScrewing1Timer	(IN:=	(eRunningState=E_GripperScrewer.eScrewing)	AND NOT tonMomentaryScrewing1Timer.Q AND 
//											mcScrewer1TorqueControl.Execute 		AND 
//											Screwing1AxisRef.NcToPlc.ActVelo < 100  AND NOT bScrewed1,
//										PT:=INT_TO_TIME(iScrewTightTime));
//	tonMomentaryScrewing2Timer	(IN:=	(eRunningState=E_GripperScrewer.eScrewing)	AND NOT tonMomentaryScrewing2Timer.Q AND 
//											mcScrewer2TorqueControl.Execute 		AND 
//											Screwing2AxisRef.NcToPlc.ActVelo < 100  AND NOT bScrewed2,
//										PT:=INT_TO_TIME(iScrewTightTime));
	
//	tonHoldingTimer			(IN:=	(eRunningState=E_GripperScrewer.eHolding ),	PT:=INT_TO_TIME(iScrewTightTime));
                  	
	tonDelayServoOn			(IN:=	(eState = E_Station.ePreparingToReady), PT:=T#20S); //bylo 1,2s
	tonResetting			(IN:=	(eState = E_Station.eResetting), 		PT:=T#4S);
	
	rtResetCommands			(CLK:=	eState = E_Station.eReady (* OR *)		,Q=>); //Triger do resetu zmienych
//	tonDelayBeforeResetLag 	(IN:=	iPreparingToReadyCase=10, 				PT:=T#10MS);

//tonFindingScrewDelay 	(IN:=	iFindingScrewCASE = 50, 				PT:=T#0MS);
//	tonStoppingCaseError	(IN:=	eState = E_Station.eStopping AND  (iStoppingCase = 30 OR iStoppingCase = 40), PT:=T#10S); 
	
	
	(*****Wyłączenie enable*****)
	IF NOT bEnable AND NOT bError THEN
		IF eState <> E_Station.eDisabled AND eState <> E_Station.ePreparingToDisable AND eState <> E_Station.eAborting AND  eState <> E_Station.eAborted THEN
			eState 				:= E_Station.ePreparingToDisable; 
		END_IF	
	END_IF

	IF eState <> E_Station.eManualMovement THEN
		
		bManualCapCatcher1								:= FALSE;
		bManualCapCatcher2								:= FALSE;
		bManualCapCatcher3								:= FALSE;
		bManualCapCatcher4					    		:= FALSE;
		bManualCapSucker1								:= FALSE;
		bManualCapSucker2								:= FALSE;
		bManualCapSucker3								:= FALSE;
		bManualCapSucker4								:= FALSE;

	END_IF


	(*****Estop*****)
	IF NOT bEstop  THEN	
		IF eState <> E_Station.eAborted AND eState <> E_Station.eAborting AND eState <> E_Station.eDisabled THEN
				iAbortingCASE		:=	0;
				eState 				:=	E_Station.eAborting; 
				
				//Jeżeli cartezjan nie jest na pozycji Ready --> wymus bazowanie
				//IF eRunningState <> E_CapPreScrewer.eReady THEN
				//	bHomingDone				:= FALSE;
				//	bHomingWithoutJiesang	:= fbBottleCatch1Station.bHomingDone;
				//END_IF
				
		END_IF
	END_IF
	
	IF NOT bRun AND bMissingCaps THEN
		bCycleNotDone				:= FALSE;
		bMissingCaps				:= FALSE;
	END_IF

	
	CASE eState OF
	/////////////////////////////	
		E_Station.eDisabled: 					// Stan nieaktywnosci (Stacja wyłączona) 
			bHomingDone				:= FALSE;
			bHomingWithoutJiesang	:= FALSE;
		
			IF bEnable  THEN
				eState 				:= E_Station.ePreparingToReady; 
			END_IF 
			
    /////////////////////////////	    
		E_Station.eAborted: 					// Stan bezpiecznego zatrzymania (po Abortingu) 
			fbGearOutAxisZ.Execute				:= CartesianZAxisRef.Status.Coupled;
			fbGearOutCatcherAxis.Execute		:= CatcherAxisRef.Status.Coupled;
		

			IF bEStop THEN
		//		bHomingDone			R= (eRunningState <> E_CapPreScrewer.eReady);
				eState 				:= E_Station.ePreparingToReady;
			END_IF
			
	/////////////////////////////	
		E_Station.eAborting:                 	// Stan bezpiecznego zatrzymywania (po EStopie)
		
			CASE iAbortingCASE OF   
				0: //Czyszczenie
					ResetCommands(); 
					iAbortingCASE	:=	iAbortingCASE	+	10;
//					iCountAborting	:=	iCountAborting	+	1;
				10: //Stop
					mcCartesianYPower.Override		:=	100;
					mcCartesianZPower.Override		:=	100;
					mcPreScrewerPower.Override		:=	100;
					mcCatcherPower.Override			:=	100;

		
					//F NOT mcHeightStop.Error AND NOT mcScrewer1Stop.Error AND NOT mcScrewer2Stop.Error THEN
					mcCartesianYStop.Execute		:=	TRUE;
					mcCartesianZStop.Execute		:=	TRUE;
					mcPreScrewerStop.Execute		:=	TRUE;
					mcCatcherStop.Execute			:= TRUE;

					iAbortingCASE					:=	iAbortingCASE	+	10;	
					//ELSE
				(*	mcHeightStop.Execute			:=	FALSE;
					mcScrewer1Stop.Execute			:=	FALSE;
					mcScrewer2Stop.Execute			:=	FALSE;
					bHeightServoPower				:=	FALSE;
					bScrewer1ServoPower				:=	FALSE;
					bScrewer2ServoPower				:=	FALSE;*)
					//END_IF	
					iCountAborting	:=	iCountAborting	+	1;						
				20: //Stop Done		
				
					IF 
						(mcCartesianYStop.Done  OR mcCartesianYStop.Error OR NOT bCartesianYServoPower) AND
						(mcCartesianZStop.Done  OR mcCartesianZStop.Error OR NOT bCartesianZServoPower) AND
						(mcCatcherStop.Done  OR mcCatcherStop.Error OR NOT bCatcherPower) AND
						(mcPreScrewerStop.Done  OR mcPreScrewerStop.Error OR NOT bPreScrewerPower)					
						 THEN
							bCartesianYServoPower		:=	FALSE;
							bCartesianZServoPower		:=	FALSE;	
							bCatcherPower				:=	FALSE;
							bPreScrewerPower			:=	FALSE;						
	
							iAbortingCASE			:=	iAbortingCASE	+	10;			
					END_IF	
					
				30: //Wyjście
					ResetCommands(); 
					eState							:=	E_Station.eAborted; 
			//		eRunningState					:=	E_CapPreScrewer.eReady;
			END_CASE
			
	/////////////////////////////			
		E_Station.eError:                 	 	// Stan błędu 	
		
			fbGearOutAxisZ.Execute				:= CartesianZAxisRef.Status.Coupled;
			mcCartesianZStop.Execute			:= CartesianZAxisRef.Status.Moving;
			
			fbGearOutCatcherAxis.Execute		:= CatcherAxisRef.Status.Coupled;
			mcCatcherStop.Execute				:= PreScrewerAxisRef.Status.Moving;


			IF bReset THEN
				eState 						:= E_Station.eResetting;
				iTestResetting					:= iTestResetting	+	1;			
			END_IF
			
	/////////////////////////////
		E_Station.eResetting:					// Stan resetowania bledu (po Errorze)
		
			diMover1VacuumRetry[1]				:= 0;
			diMover1VacuumRetry[2]				:= 0;
			diMover1VacuumRetry[3]				:= 0;
			diMover1VacuumRetry[4]				:= 0;
			fbVirtualAxis.Reset(bExecute := fbVirtualAxis.bError);	

			//Procedura obsługi resetu w zależności od błędu
			CASE udiErrorID OF
			
				//Error 2 - BŁĄD SERWA WÓZKA 1
				//Error 3 - BŁĄD SERWA WÓZKA 2			
				0, 1129..1132, 1151..1159:	

					CASE iErrorResseting2 OF
					0:
						IF mcCartesianYPower.Status THEN
							bCartesianYServoPower 	:= FALSE;
						END_IF
						
						IF mcCartesianZPower.Status THEN
							bCartesianZServoPower 	:= FALSE;
						END_IF

						IF mcCatcherPower.Status THEN
							bCatcherPower			:= FALSE;
						END_IF
						
						IF mcPreScrewerPower.Status THEN
							bPreScrewerPower 		:= FALSE;
						END_IF
		
						fbCartesianYHardReset		(Execute:=TRUE,	Axis:=CartesianYAxisRef);
						fbCartesianZHardReset		(Execute:=TRUE,	Axis:=CartesianZAxisRef);
						fbPreScrewerHardReset		(Execute:=TRUE,	Axis:=PreScrewerAxisRef);
						fbCatcherHardReset			(Execute:=TRUE,	Axis:=CatcherAxisRef);
						mcCartesianYSoftReset		(Execute:=TRUE,	Axis:=CartesianYAxisRef); 
						mcCartesianZSoftReset		(Execute:=TRUE,	Axis:=CartesianZAxisRef);
						mcPreScrewerSoftReset		(Execute:=TRUE,	Axis:=PreScrewerAxisRef);
						mcCatcherSoftReset			(Execute:=TRUE,	Axis:=CatcherAxisRef);
						fbVirtualAxis.Reset(bExecute := fbVirtualAxis.bError);						
		
						IF bEnable THEN
							bCartesianYServoPower 	:= TRUE;
							bCartesianzServoPower 	:= TRUE;
							bPreScrewerPower		:= TRUE;
							bCatcherPower			:= TRUE;	
						END_IF
						

						IF 
						( NOT fbCartesianYHardReset.Busy AND NOT mcCartesianYSoftReset.Busy AND (mcCartesianYPower.Status OR NOT bEnable) AND NOT CartesianYAxisRef.Status.Error ) AND
						( NOT fbCartesianZHardReset.Busy AND NOT mcCartesianZSoftReset.Busy AND (mcCartesianZPower.Status OR NOT bEnable) AND NOT CartesianZAxisRef.Status.Error ) AND
						( NOT fbPreScrewerHardReset.Busy AND NOT mcPreScrewerSoftReset.Busy AND (mcPreScrewerPower.Status OR NOT bEnable) AND NOT PreScrewerAxisRef.Status.Error ) AND
						( NOT fbCatcherHardReset.Busy AND NOT mcCatcherSoftReset.Busy AND (mcCatcherPower.Status OR NOT bEnable) AND NOT CatcherAxisRef.Status.Error AND (NOT fbVirtualAxis.bError OR NOT VirtualEna))
						
						THEN
							fbCartesianYHardReset		(Execute:=FALSE,	Axis:=CartesianYAxisRef);
							fbCartesianZHardReset		(Execute:=FALSE,	Axis:=CartesianZAxisRef);
							fbPreScrewerHardReset		(Execute:=FALSE,	Axis:=PreScrewerAxisRef);
							fbCatcherHardReset			(Execute:=FALSE,	Axis:=CatcherAxisRef);
							mcCartesianYSoftReset		(Execute:=FALSE,	Axis:=CartesianYAxisRef); 
							mcCartesianZSoftReset		(Execute:=FALSE,	Axis:=CartesianZAxisRef);
							mcPreScrewerSoftReset		(Execute:=FALSE,	Axis:=PreScrewerAxisRef);
							mcCatcherSoftReset			(Execute:=FALSE,	Axis:=CatcherAxisRef);		
							


							bError								:=	FALSE;
							iErrorResseting2					:=	0;	
							udiCartesianXServoErrorNr			:=	0;
							udiCartesianZServoErrorNr			:=	0;
							sErrorDescription					:=	'';
							sErrorDescription2					:=	'';

							udiErrorID							:=	0;
						END_IF	
					END_CASE
				
				1133..1141:
				//fbCartesianZHardReset(Execute:=CartesianZAxisRef.Status.Error,	Axis:=CartesianZAxisRef);
				//mcCartesianZSoftReset(Execute:=CartesianZAxisRef.Status.Error,	Axis:=CartesianZAxisRef);	
				//
				//IF (NOT CartesianZAxisRef.Status.Error AND NOT fbCartesianZHardReset.Busy
				//	AND NOT mcCartesianZSoftReset.Busy AND mcCartesianZPower.Status) THEN
				//		mcCartesianZMoveAbsolute.Execute		:= TRUE;		
				//		mcCartesianZMoveAbsolute.Position		:= 450.0;
				//		mcCartesianZMoveAbsolute.Acceleration	:= 1000.0;
				//		mcCartesianZMoveAbsolute.Deceleration	:= 1000.0;
				//		mcCartesianZMoveAbsolute.Velocity		:= 15.0;
				//END_IF	
				//
				//IF mcCartesianZMoveAbsolute.Done THEN
					bStrawCatcherActuatorIn						:= FALSE;
					bStrawCatcherActuatorOut					:= FALSE;
					mcCartesianZMoveAbsolute.Execute			:= FALSE;
					bError										:= FALSE;
					iErrorResseting2							:= 0;	
					udiCartesianXServoErrorNr					:= 0;
					udiCartesianZServoErrorNr					:= 0;
					sErrorDescription							:= '';
					sErrorDescription2							:= '';
                	                                    		   
					udiErrorID									:= 0;	
				//END_IF	
	
			
				//Error 6 - BŁAD POZYCJI MINIMALNEJ PODNOŚNIKA 
				6:
					IF NOT fbStrawCatcherLift.bError THEN
						bError										:= FALSE;						
					END_IF			
				1142..1150:
				
					diMover2VacuumRetry[1]				:= 0;
					diMover2VacuumRetry[2]				:= 0;
					diMover2VacuumRetry[3]				:= 0;
					diMover2VacuumRetry[4]				:= 0;
					bError								:=	FALSE;
					sErrorDescription					:=	'';
					sErrorDescription2					:=	'';
				ELSE
					bError								:=	FALSE;	
			END_CASE	
			
			IF NOT bError THEN
				udiErrorID 						:=	0;
   				sErrorDescription 				:=	'';                       			
				eState 							:=	E_Station.ePreparingToReady;
			ELSIF tonResetting.Q THEN     
				ResetCommands();       	
				eState 							:=	E_Station.eError;
			END_IF
        
	/////////////////////////////
		E_Station.eManualMovement:     			// Stan ruchów manualnych  
		
			IF bHoming THEN
				eState 				:= E_Station.eHoming; 
			END_IF
       
			ManualMovements(); 
			//Wyjście z trybu serwisowego
			IF NOT bManualMovement THEN
					//bManualGripper1				:=	FALSE;
					//bManualGripper2				:=	FALSE;		
	

			
					mcCartesianYPower.Override		:= 100;
					mcCartesianZPower.Override		:= 100;
					mcPreScrewerPower.Override		:= 100;
					mcCatcherPower.Override			:= 100;
//					IF
//						Height1AxisRef.NcToPlc.ActPos	<=	lrHeightReadyPosition OR
//						Height2AxisRef.NcToPlc.ActPos	<=	lrHeightReadyPosition
//					THEN
//						mcHeight1MoveAbsolute.Execute		:=	TRUE;
//						mcHeight1MoveAbsolute.Position		:=	lrHeightReadyPosition;
						
//						mcHeight2MoveAbsolute.Execute		:=	TRUE;
//						mcHeight2MoveAbsolute.Position		:=	lrHeightReadyPosition;
//						IF mcHeight1MoveAbsolute.Done AND mcHeight2MoveAbsolute.Done THEN
//							mcHeight1MoveAbsolute.Execute	:=	FALSE;
//							mcHeight2MoveAbsolute.Execute	:=	FALSE;
//							eState							:=	E_Station.eReady;
//						END_IF	
//					ELSE
							eState							:=	E_Station.eReady;
//					END_IF	
			END_IF

	/////////////////////////////
		E_Station.eHoming:						// Stan bazowania 

			Homing();
			IF NOT bHoming THEN
			  	eState							:=	E_Station.ePreparingToReady;
			   	mcCartesianYManualMove.JogBackwards		:=FALSE;
				mcCartesianZManualMove.JogBackwards		:=FALSE;
				mcPreScrewerManualMove.JogBackwards		:=FALSE;
				mcCatcherManualMove.JogBackwards		:=FALSE;
				
				mcCartesianYManualMove.JogForward		:=FALSE;
				mcCartesianZManualMove.JogForward		:=FALSE;
				mcPreScrewerManualMove.JogForward		:=FALSE;
				mcCatcherManualMove.JogForward			:=FALSE;			
			END_IF		
			
	/////////////////////////////
		E_Station.eHomingDone:                  // Stan wykonania bazowania 
		
			bAdvancedHoming							:= FALSE;
			mcCartesianYManualMove.JogBackwards		:= FALSE;
			mcCartesianZManualMove.JogBackwards		:= FALSE;
			mcPreScrewerManualMove.JogBackwards		:= FALSE;
			mcCatcherManualMove.JogBackwards		:= FALSE;
			                                           
			mcCartesianYManualMove.JogForward		:= FALSE;
			mcCartesianZManualMove.JogForward		:= FALSE;
			mcPreScrewerManualMove.JogForward		:= FALSE;
			mcCatcherManualMove.JogForward			:= FALSE;
			                                           
			bHomingDone								:= TRUE;
			IF NOT bHoming THEN                 	
				eRunningState						:= E_CapPreScrewer.eReady;
			   	eState								:= E_Station.eReady;
			END_IF
			
	/////////////////////////////
		E_Station.ePreparingToReady:            // Stan przygotowywania do gotowosci (zawsze przed Ready)  

		//	IF tonDelayServoOn.Q(*bySafetyStateScrewer1.0 AND bySafetyStateScrewer2.0 AND bySafetyStateHightServo.0 *)THEN
				bCartesianYServoPower	:= nAxisYSafetyState.0;	// Przy pierwszym uruchomieniu Ustawienia Fabryczne robimy na wartość maksymalną
				bCartesianZServoPower	:= nAxisZSafetyState.0;	// Przy pierwszym uruchomieniu Ustawienia Fabryczne robimy na wartość maksymalną
				bPreScrewerPower		:= nAxisScrewSafetyState.0;
				bCatcherPower			:= nAxisCatcherSafetyState.0;
//				bStrawCatcherLiftEnable	:= TRUE;
		//	END_IF	
			
			IF mcCartesianYPower.Status AND mcCartesianZPower.Status AND mcPreScrewerPower.Status AND mcCatcherPower.Status  THEN 

				IF NOT bAxisYInPosition OR NOT bAxisZInPosition OR NOT bCartesianInReadyPos  THEN
					bHomingDone							:= FALSE;
					bHomingWithoutJiesang				:= fbStrawCatcherLift.bHomingDone;
				END_IF	
				 		
				eState									:=	E_Station.eReady;
			END_IF
			
         	IF bIgnoreError THEN
				eState										:=	E_Station.eReady;
			END_IF
	
	/////////////////////////////
		E_Station.ePreparingToDisable:          // Stan przygotowywania do nieaktywnosci (po wyłączeniu Enable) 
  
			bCartesianYServoPower	:= TRUE;	// Przy pierwszym uruchomieniu Ustawienia Fabryczne robimy na wartość maksymalną
			bCartesianZServoPower	:= TRUE;	// Przy pierwszym uruchomieniu Ustawienia Fabryczne robimy na wartość maksymalną
			bPreScrewerPower		:= TRUE;
			bCatcherPower			:= TRUE;
			
			eRunningState					:=	E_CapPreScrewer.eReady;		//Dodane
			PreparingToDisable();

         	IF bIgnoreError THEN
				eState:=E_Station.eDisabled;
			END_IF
			
	/////////////////////////////
		E_Station.eReady:						// Stan gotowosci 
		
		//Detekcja utraconej nasadki
			GVL_UVFF.ftVacuumSensor1(CLK := tonSuckedOk[1].Q);
			GVL_UVFF.ftVacuumSensor2(CLK := tonSuckedOk[2].Q);
			GVL_UVFF.ftVacuumSensor3(CLK := tonSuckedOk[3].Q);
			GVL_UVFF.ftVacuumSensor4(CLK := tonSuckedOk[4].Q);
		
				//Jeżeli utracimy nasadkę--> wyłącz ssawkę
			//bCapSucker[1]					R= GVL.ftVacuumSensor1.Q;
			//bCapSucker[2]					R= GVL.ftVacuumSensor2.Q;
			//bCapSucker[3]					R= GVL.ftVacuumSensor3.Q;
			//bCapSucker[4]					R= GVL.ftVacuumSensor4.Q;
			
			bEnableLift					:= FALSE;
		
		//Zdejmuję HomingDone gdy utracę bodaj jedną nasadkę lub Jiesang nie jest zbazowany
			//IF (*bAnyCapLost OR*) (NOT fbBottleCatch1Station.bHomingDone AND NOT bManualMovement) THEN
			//	bHomingDone					:= FALSE;
			//	bHomingWithoutJiesang		:= fbBottleCatch1Station.bHomingDone;
			//END_IF
		
			(*Skasowanie wszystkich komend*)
			IF rtResetCommands.Q THEN	
				ResetCommands();	
			END_IF
			
			IF bPreRun THEN
				eState						:= E_Station.eStarting;
			END_IF
			
			IF bRun AND NOT bCycleDone (*AND NOT bCycleNotDone*) AND bHomingDone THEN
				eState 						:= E_Station.eRunning; 
			END_IF
			IF bHoming THEN
				eState 						:= E_Station.eHoming; 
			END_IF
			
			IF NOT bRun THEN
				GVL_VIS.bCapSorterPreScrewerBottleCatcherCatch	:= FALSE;
				bPlaceDone										:= FALSE;
				bCycleDone 										:= FALSE;		
			END_IF
			
			IF bManualMovement THEN
				//Jeśli przejście w tryb ruchów manualnych przepisz wszystkie stany siłowników sterowanych przez moduł
				//aby zapobiec ewentualnym kolizjom po wejściu w tryb serwisowy
				//Ruchy manualne siłownika na wózku	
				bManualCapSucker1							:= bCapSucker[1];	
				bmanualCapSucker2							:= bCapSucker[2];	
				bManualCapSucker3							:= bCapSucker[3];	
				bManualCapSucker4							:= bCapSucker[4];	
				                          	    		                 
				bManualCapBlower1							:= bCapBlower1;	
				bManualCapBlower2							:= bCapBlower2;	
				bManualCapBlower3							:= bCapBlower3;	
				bManualCapBlower4							:= bCapBlower4;	
				                          		    	                 
				bManualCapCatcher1							:= bCapCatcher1;
				bManualCapCatcher2							:= bCapCatcher2;
				bManualCapCatcher3							:= bCapCatcher3;
				bManualCapCatcher4					    	:= bCapCatcher4;
				                                        	
				bManualStrawCatchersOpen					:= bStrawCatchersOpen;
				bManualStrawCatchersClose					:= bStrawCatchersClose;	                                            	
				                                        	
			    bManualStrawCatcherActuatorOut 				:= bStrawCatcherActuatorOut;
			    bManualStrawCatcherActuatorIn 				:= bStrawCatcherActuatorIn;
				
				bHomingWithoutJiesang						:= fbStrawCatcherLift.bHomingDone;
				
				eState 										:=	E_Station.eManualMovement; 

			END_IF
			
	/////////////////////////////
		E_Station.eStopping:					// Stan zatrzymywania 
			
			RunningCam();//RunningWithFlyingSaw();				//Running();
			
					IF bStopAllowed THEN
						eState 								:=	E_Station.eReady;
					END_IF

				
	/////////////////////////////
		E_Station.eStarting:                  	// Stan uruchamiania (po Ready)				
		
		IF 	eRunningState = E_CapPreScrewer.eReady THEN	//Jeżeli jesteśmy na poz. ready--> sprawdź i dojedź do pozycji home
				//Dojazd do poz top		                                                    	
			mcCartesianZMoveAbsolute.Execute						:= NOT bAxisZInTopPos;		
			mcCartesianZMoveAbsolute.Position						:= stParameters.lrTopZPosition;
			mcCartesianZMoveAbsolute.Acceleration					:= 500.0;
			mcCartesianZMoveAbsolute.Deceleration					:= 500.0;
			mcCartesianZMoveAbsolute.Velocity						:= 50;
			                                        				
			//najpierw os Z potem winda chwytakow   				
			mcCatcherMoveAbsolute.Execute							:= NOT bAxisStrawCatcherHomePos AND bAxisZInTopPos;		
			mcCatcherMoveAbsolute.Position							:= stParameters.lrCatcherCatchingPosition;
			mcCatcherMoveAbsolute.Acceleration						:= 300.0;
			mcCatcherMoveAbsolute.Deceleration						:= 300.0;
			mcCatcherMoveAbsolute.Velocity							:= 30;
			                                        				
			mcCartesianYMoveAbsolute.Execute						:= NOT bAxisYInHomePos AND bAxisZInTopPos;
			mcCartesianYMoveAbsolute.Position						:= stParameters.lrPickYPosition;
			mcCartesianYMoveAbsolute.Acceleration					:= 500.0;
			mcCartesianYMoveAbsolute.Deceleration					:= 500.0;
			mcCartesianYMoveAbsolute.Velocity						:= 50; 
			                                                    	
			IF bAxisZInTopPos THEN
				GVL_VIS.bCapSorterPreScrewerCatchStationHoming			:= NOT fbStrawCatcherLift.bHomingDone;
				GVL_VIS.bCapSorterPreScrewerCatcherStationHeightSet		:= NOT GVL_VIS.bCapSorterPreScrewerCatchStationHoming AND NOT bStrawCatcherLiftInHomePos;
				bEnableLift												:= TRUE;
			END_IF
    		
				IF 	bCartesianInTopPos AND bStrawCatcherLiftInHomePos THEN
					mcCartesianZMoveAbsolute.Execute              	:= FALSE;
					mcCatcherMoveAbsolute.Execute                 	:= FALSE;
					mcCartesianYMoveAbsolute.Execute              	:= FALSE;
					GVL_VIS.bCapSorterPreScrewerCatchStationHoming	:= FALSE;
					eState											:= E_Station.eRunning; 
				END_IF
		ELSE
			eState							:= E_Station.eRunning; 
			bEnableLift						:= TRUE;	
		END_IF	
					
			
	/////////////////////////////
		E_Station.eRunning:               		// Stan wykonywania cyklu (po Startingu), w tym stanie osobny
		
 			IF bRun THEN
				IF bSimulationEna THEN
					Simulation();
				ELSE	
					RunningCam();	//RunningWithFlyingSaw();				//Running();
				END_IF
				
				
			ELSIF NOT bPreRun THEN
				bBottleCatcherCatchTemp		:= FALSE;
				eState 				 		:= E_Station.eStopping;		
			END_IF
				
			
	/////////////////////////////	
		E_Station.eDone:
		
			IF bCycleDone THEN (*Cykl zakończony*)
				bBottleCatcherCatchTemp		:= FALSE;
			END_IF	
			
			IF NOT bPreRun  AND bStopAllowed THEN					(*Przerywanie cyklu*)
				bBottleCatcherCatchTemp		:= FALSE;
				eState 				 		:= E_Station.eStopping;	
			ELSIF NOT bRun THEN
				GVL_VIS.bCapSorterPreScrewerBottleCatcherCatch	:= FALSE;
				bPlaceDone										:= FALSE;
				bCycleDone 										:= FALSE;	
				eState 				 							:= E_Station.eRunning;	
			END_IF
		
		
		
	END_CASE

	
//IF (ABS(GVL_VIS.lrCapSorterPreScrewerCatcherStationHeightCV-stParameters.lrCatcherHightSV) > 2) AND
//	(eState = E_Station.eStarting OR eState = E_Station.ePreparingToReady) THEN
//			GVL_VIS.bCapSorterPreScrewerCatcherStationHeightSet 				:= TRUE;
//ELSIF ABS(GVL_VIS.lrCapSorterPreScrewerCatcherStationHeightCV-stParameters.lrCatcherHightSV) < 2 THEN
//			GVL_VIS.bCapSorterPreScrewerCatcherStationHeightSet 				:= FALSE;	
//END_IF
END_ACTION

ACTION ErrorHandling:
//CZYTANIE STATUSÓW
CartesianYAxisRef.ReadStatus();
CartesianZAxisRef.ReadStatus();
CatcherAxisRef.ReadStatus();
PreScrewerAxisRef.ReadStatus();
//Czasówki od siłowników
tonErrorStrawCatcherIn(IN:= bStrawCatcherActuatorIn AND NOT bStrawCatcherIn,PT:=T#1000MS);
tonErrorStrawCatcherOut(IN:= bStrawCatcherActuatorOut AND NOT bStrawCatcherOut,PT:=T#1000MS);



//**********************LISTA BŁĘDÓW******************************
bStateError	:= (eState=E_Station.eError) OR (eState=E_Station.eResetting) OR NOT bEstop OR bIgnoreError;

//PreparingToDisable i StateError ze względu na wciśnięcie EStopa podczas wyłączania i pojawienie się blędu
IF bEnable OR eState=E_Station.ePreparingToDisable THEN
	


	//Error 1 - BŁĄD SERWA POZIOMEGO X
	IF (CartesianYAxisRef.Status.Error OR mcCartesianYMoveAbsolute.Error) AND NOT arrFbAllarm[0].bActive THEN
		sAxisAlarm := CONCAT(UDINT_TO_STRING(CartesianYAxisRef.Status.ErrorID),F_AxErrMsg(CartesianYAxisRef.Status.ErrorID));
		arrFbAllarm[0].ipArguments.Clear().AddString(sAxisAlarm);		
		arrFbAllarm[0].Raise(nTimeStamp := 0);		
		udiErrorID							:=	1129;
		udiCartesianXServoErrorNr			:=	CartesianYAxisRef.Status.ErrorID;
		sErrorDescription					:=	'Błąd napędu poziomego Y. Błąd NC:';
		sErrorDescription2					:=	F_AX8xErrMsg(TO_UINT(udiCartesianXServoErrorNr));
	ELSIF NOT CartesianYAxisRef.Status.Error AND NOT mcCartesianYMoveAbsolute.Error AND eState = E_Station.eResetting AND arrFbAllarm[0].bActive THEN
			arrFbAllarm[0].Clear(nTimeStamp := 0, bResetConfirmation := FALSE);
	END_IF;
	
	//Error 2 - BŁĄD SERWA PIONOWEGO Z
	IF (CartesianZAxisRef.Status.Error OR mcCartesianZMoveAbsolute.Error) AND NOT arrFbAllarm[1].bActive THEN
		sAxisAlarm := CONCAT(UDINT_TO_STRING(CartesianZAxisRef.Status.ErrorID),F_AxErrMsg(CartesianZAxisRef.Status.ErrorID));
		arrFbAllarm[1].ipArguments.Clear().AddString(sAxisAlarm);		
		arrFbAllarm[1].Raise(nTimeStamp := 0);		
		udiErrorID							:=	1130;
		udiCartesianZServoErrorNr			:=	CartesianZAxisRef.Status.ErrorID;
		sErrorDescription					:=	'Błąd napędu podnoszenia Z. Błąd NC:';
		sErrorDescription2					:=	F_AX8xErrMsg(TO_UINT(udiCartesianZServoErrorNr));
	ELSIF NOT CartesianZAxisRef.Status.Error AND NOT mcCartesianZMoveAbsolute.Error AND eState = E_Station.eResetting AND arrFbAllarm[1].bActive THEN
			arrFbAllarm[1].Clear(nTimeStamp := 0, bResetConfirmation := FALSE);
	END_IF;
	
	//Error 3 - BŁĄD SERWA PIONOWEGO UCHWYTU SŁOMEK
	IF (CatcherAxisRef.Status.Error OR mcCatcherMoveAbsolute.Error) AND NOT arrFbAllarm[2].bActive THEN		
		sAxisAlarm := CONCAT(UDINT_TO_STRING(CatcherAxisRef.Status.ErrorID),F_AxErrMsg(CatcherAxisRef.Status.ErrorID));
		arrFbAllarm[2].ipArguments.Clear().AddString(sAxisAlarm);		
		arrFbAllarm[2].Raise(nTimeStamp := 0);		
		udiErrorID							:=	1131;
		udiCatcherServoErrorNr				:=	CatcherAxisRef.Status.ErrorID;
		sErrorDescription					:=	'Błąd napędu podnoszenia chwytaka słomek. Błąd NC:';
		sErrorDescription2					:=	F_AX8xErrMsg(TO_UINT(udiCatcherServoErrorNr));
	ELSIF NOT CatcherAxisRef.Status.Error AND NOT  mcCatcherMoveAbsolute.Error AND eState = E_Station.eResetting AND arrFbAllarm[2].bActive THEN
			arrFbAllarm[2].Clear(nTimeStamp := 0, bResetConfirmation := FALSE);
	END_IF;
	
	//Error 4 - BŁĄD SERWA OBROTOWEGO
	IF (PreScrewerAxisRef.Status.Error OR mcPreScrewerMoveAbsolute.Error OR bTestError) AND NOT arrFbAllarm[3].bActive THEN
		sAxisAlarm := CONCAT(UDINT_TO_STRING(PreScrewerAxisRef.Status.ErrorID),F_AxErrMsg(PreScrewerAxisRef.Status.ErrorID));
		arrFbAllarm[3].ipArguments.Clear().AddString(sAxisAlarm);		
		arrFbAllarm[3].Raise(nTimeStamp := 0);		
		udiErrorID							:=	1132;
		udiPreScrewerServoErrorNr			:=	PreScrewerAxisRef.Status.ErrorID;
		sErrorDescription					:=	'Błąd napędu zakręcania. Błąd NC:';
		sErrorDescription2					:=	F_AX8xErrMsg(TO_UINT(udiPreScrewerServoErrorNr));
	ELSIF NOT PreScrewerAxisRef.Status.Error AND NOT  mcPreScrewerMoveAbsolute.Error AND eState = E_Station.eResetting AND arrFbAllarm[3].bActive THEN
			arrFbAllarm[3].Clear(nTimeStamp := 0, bResetConfirmation := FALSE);
	END_IF;
	
	IF PreScrewerAxisRef.Status.Error THEN
		GVL_UVFF.diTest1	:= GVL_UVFF.diTest1 + 1;
	END_IF
	
	IF mcPreScrewerMoveAbsolute.Error THEN
		GVL_UVFF.diTest2	:= GVL_UVFF.diTest2 + 1;
	END_IF
	
	IF mcPreScrewerMoveRelative.Error THEN
		GVL_UVFF.diTesy3	:= GVL_UVFF.diTesy3 + 1;
	END_IF
	
	IF bTestError THEN
		GVL_UVFF.diTest4	:= GVL_UVFF.diTest4 + 1;
	END_IF	
	
	
	
	
	
	//Error 5A - BŁĄD PRZEKROCZENIE CZASU DZIAŁANIA SIŁOWNIKA CHWYTAKÓW SŁOMEK
	IF tonErrorStrawCatcherOut.Q AND NOT arrFbAllarm[4].bActive THEN
		arrFbAllarm[4].Raise(nTimeStamp := 0);	
		udiErrorID							:=	1133;
		udiPreScrewerServoErrorNr			:=	PreScrewerAxisRef.Status.ErrorID;
		sErrorDescription					:=	'Błąd siłownika chwytaków słomek | Zablokowany wysów';
		sErrorDescription2					:=	'';
	ELSIF NOT tonErrorStrawCatcherOut.Q AND eState = E_Station.eResetting AND arrFbAllarm[4].bActive THEN
			arrFbAllarm[4].Clear(nTimeStamp := 0, bResetConfirmation := FALSE);
	END_IF;
	
	//Error 5B - BŁĄD PRZEKROCZENIE CZASU DZIAŁANIA SIŁOWNIKA CHWYTAKÓW SŁOMEK
	IF tonErrorStrawCatcherIn.Q AND NOT arrFbAllarm[5].bActive THEN
		arrFbAllarm[5].Raise(nTimeStamp := 0);	
		udiErrorID							:=	1134;
		udiPreScrewerServoErrorNr			:=	PreScrewerAxisRef.Status.ErrorID;
		sErrorDescription					:=	'Błąd siłownika chwytaków słomek | Zablokowane cofnięcie';
		sErrorDescription2					:=	'';
	ELSIF NOT tonErrorStrawCatcherIn.Q AND eState = E_Station.eResetting AND arrFbAllarm[5].bActive THEN
			arrFbAllarm[5].Clear(nTimeStamp := 0, bResetConfirmation := FALSE);
	END_IF;
	
	//Error 6 - Blad podnosnika Jiecang - brak zasilania lub zablokowany mechanicznie
	IF fbStrawCatcherLift.bError AND fbStrawCatcherLift.nErrorNr = 1 AND NOT arrFbAllarm[6].bActive THEN
		arrFbAllarm[6].Raise(nTimeStamp := 0);	
    	udiErrorID				:= 1135;
    	sErrorDescription		:= 'Błąd podnosnika lub brak zasilania';
    	sErrorDescription2		:= ' ';
	ELSIF NOT fbStrawCatcherLift.bError AND eState = E_Station.eResetting AND arrFbAllarm[6].bActive THEN
			arrFbAllarm[6].Clear(nTimeStamp := 0, bResetConfirmation := FALSE);
	END_IF;
		

	//Error 6 - Blad podnosnika Jiecang - prak zasilania lub zablokowany mechanicznie
	IF fbStrawCatcherLift.bError AND fbStrawCatcherLift.nErrorNr = 2 AND NOT arrFbAllarm[7].bActive THEN
		arrFbAllarm[7].Raise(nTimeStamp := 0);
    	udiErrorID				:= 1136;
    	sErrorDescription		:= 'Błąd podnosnika  - wartość zadana jest większa od wartości maksymalnej';
    	sErrorDescription2		:= ' ';
	ELSIF NOT fbStrawCatcherLift.bError AND eState = E_Station.eResetting AND arrFbAllarm[7].bActive THEN
			arrFbAllarm[7].Clear(nTimeStamp := 0, bResetConfirmation := FALSE);
	END_IF;
	
	
	//Error 6 - Blad podnosnika Jiecang - prak zasilania lub zablokowany mechanicznie
	IF  fbStrawCatcherLift.bError AND fbStrawCatcherLift.nErrorNr = 3 AND NOT arrFbAllarm[8].bActive THEN
		arrFbAllarm[8].Raise(nTimeStamp := 0);
    	udiErrorID				:= 1137;
    	sErrorDescription		:= 'Błąd podnosnika - wartość zadana jest mniejsza od wartości minimalnej';
    	sErrorDescription2		:= ' ';
	ELSIF NOT fbStrawCatcherLift.bError AND eState = E_Station.eResetting AND arrFbAllarm[8].bActive THEN
			arrFbAllarm[8].Clear(nTimeStamp := 0, bResetConfirmation := FALSE);
	END_IF;
	
		//Error 11 - Blad Kolizja	
	IF  rtCollisionError.Q AND NOT arrFbAllarm[13].bActive THEN
		arrFbAllarm[13].Raise(nTimeStamp := 0);
    	udiErrorID				:= 1142;
    	sErrorDescription		:= 'Kolizja kartezjana z transporterem nakrętek | Zbazuj stacje wkładania nakrętek';
    	sErrorDescription2		:= '';
	ELSIF NOT  rtCollisionError.Q AND eState = E_Station.eResetting AND arrFbAllarm[13].bActive THEN
			arrFbAllarm[13].Clear(nTimeStamp := 0, bResetConfirmation := FALSE);
	END_IF;

		//Przekroczona ilość prób pobrania nasadki, mówer1, słot1
	IF diMover1VacuumRetry[1] >= 3  AND NOT arrFbAllarm[14].bActive THEN
		arrFbAllarm[14].Raise(nTimeStamp := 0);
    	udiErrorID				:= 1143;
    	sErrorDescription		:= 'Przekroczona ilość prób pobrania nasadki, wózek1, slot1';
    	sErrorDescription2		:= '';
	ELSIF diMover1VacuumRetry[1] < 3 AND eState = E_Station.eResetting AND arrFbAllarm[14].bActive THEN
			arrFbAllarm[14].Clear(nTimeStamp := 0, bResetConfirmation := FALSE);
	END_IF;
	
	IF diMover1VacuumRetry[2] >= 3  AND NOT arrFbAllarm[15].bActive THEN
		arrFbAllarm[15].Raise(nTimeStamp := 0);
    	udiErrorID				:= 1144;
    	sErrorDescription		:= 'Przekroczona ilość prób pobrania nasadki, wózek1, slot2';
    	sErrorDescription2		:= '';
	ELSIF diMover1VacuumRetry[2] < 3 AND eState = E_Station.eResetting AND arrFbAllarm[15].bActive THEN
			arrFbAllarm[15].Clear(nTimeStamp := 0, bResetConfirmation := FALSE);
	END_IF;

	IF diMover1VacuumRetry[3] >= 3  AND NOT arrFbAllarm[16].bActive THEN
		arrFbAllarm[16].Raise(nTimeStamp := 0);
    	udiErrorID				:= 1145;
    	sErrorDescription		:= 'Przekroczona ilość prób pobrania nasadki, wózek1, slot3';
    	sErrorDescription2		:= '';
	ELSIF diMover1VacuumRetry[3] < 3 AND eState = E_Station.eResetting AND arrFbAllarm[16].bActive THEN
			arrFbAllarm[16].Clear(nTimeStamp := 0, bResetConfirmation := FALSE);
	END_IF;
	
	IF diMover1VacuumRetry[4] >= 3  AND NOT arrFbAllarm[17].bActive THEN
		arrFbAllarm[17].Raise(nTimeStamp := 0);
    	udiErrorID				:= 1146;
    	sErrorDescription		:= 'Przekroczona ilość prób pobrania nasadki, wózek1, slot4';
    	sErrorDescription2		:= '';
	ELSIF diMover1VacuumRetry[4] < 3 AND eState = E_Station.eResetting AND arrFbAllarm[17].bActive THEN
			arrFbAllarm[17].Clear(nTimeStamp := 0, bResetConfirmation := FALSE);
	END_IF;
	
			//Przekroczona ilość prób pobrania nasadki, mówer2, słot1
	IF diMover2VacuumRetry[1] >= 3  AND NOT arrFbAllarm[18].bActive THEN
		arrFbAllarm[18].Raise(nTimeStamp := 0);
    	udiErrorID				:= 1147;
    	sErrorDescription		:= 'Przekroczona ilość prób pobrania nasadki, wózek2, slot1';
    	sErrorDescription2		:= '';
	ELSIF diMover2VacuumRetry[1] < 3 AND eState = E_Station.eResetting AND arrFbAllarm[18].bActive THEN
			arrFbAllarm[18].Clear(nTimeStamp := 0, bResetConfirmation := FALSE);
	END_IF;
	
	IF diMover2VacuumRetry[2] >= 3  AND NOT arrFbAllarm[19].bActive THEN
		arrFbAllarm[19].Raise(nTimeStamp := 0);
    	udiErrorID				:= 1148;
    	sErrorDescription		:= 'Przekroczona ilość prób pobrania nasadki, wózek2, slot2';
    	sErrorDescription2		:= '';
	ELSIF diMover2VacuumRetry[2] < 3 AND eState = E_Station.eResetting AND arrFbAllarm[19].bActive THEN
			arrFbAllarm[19].Clear(nTimeStamp := 0, bResetConfirmation := FALSE);
	END_IF;

	IF diMover2VacuumRetry[3] >= 3  AND NOT arrFbAllarm[20].bActive THEN
		arrFbAllarm[20].Raise(nTimeStamp := 0);
    	udiErrorID				:= 1149;
    	sErrorDescription		:= 'Przekroczona ilość prób pobrania nasadki, wózek2, slot3';
    	sErrorDescription2		:= '';
	ELSIF diMover2VacuumRetry[3] < 3 AND eState = E_Station.eResetting AND arrFbAllarm[20].bActive THEN
			arrFbAllarm[20].Clear(nTimeStamp := 0, bResetConfirmation := FALSE);
	END_IF;
	
	IF diMover2VacuumRetry[4] >= 3  AND NOT arrFbAllarm[21].bActive THEN
		arrFbAllarm[21].Raise(nTimeStamp := 0);
    	udiErrorID				:= 1150;
    	sErrorDescription		:= 'Przekroczona ilość prób pobrania nasadki, wózek2, slot4';
    	sErrorDescription2		:= '';
	ELSIF diMover2VacuumRetry[4] < 3 AND eState = E_Station.eResetting AND arrFbAllarm[21].bActive THEN
			arrFbAllarm[21].Clear(nTimeStamp := 0, bResetConfirmation := FALSE);
	END_IF;

	IF NOT arrFbAllarm[22].bActive AND (fbVirtualAxis.bErrorFB  OR fbVirtualAxis.bError) THEN	
		sAxisAlarm := CONCAT(UDINT_TO_STRING(fbVirtualAxis.nErrorId),F_AxErrMsg(fbVirtualAxis.nErrorId));
		arrFbAllarm[22].ipArguments.Clear().AddString(sAxisAlarm);		
		arrFbAllarm[22].Raise(nTimeStamp := 0);	
		udiErrorID							:=	1151;
		sErrorDescription					:=	'Błąd wirtualnej osi:';
		sErrorDescription2					:=	F_AX8xErrMsg(TO_UINT(fbVirtualAxis.nErrorId));
	ELSIF NOT fbVirtualAxis.bError AND NOT  fbVirtualAxis.bErrorFB AND eState = E_Station.eResetting AND arrFbAllarm[22].bActive THEN
			arrFbAllarm[22].Clear(nTimeStamp := 0, bResetConfirmation := FALSE);
	END_IF;
	
	IF (fbVirtualAxis.pSetPos.Error OR fbVirtualAxis.pSetPos.CommandAborted) AND NOT arrFbAllarm[23].bActive THEN
		arrFbAllarm[23].ipArguments.Clear().AddUDInt(fbVirtualAxis.pSetPos.ErrorID);		
		arrFbAllarm[23].Raise(nTimeStamp := 0);		
    	udiErrorID							:= 1152;
    	udiErrorID							:= udiErrorID + iStationIndex;
    	sErrorDescription					:= CONCAT('Błąd wirtualnej osi', UDINT_TO_STRING(fbVirtualAxis.pSetPos.ErrorID));
    	sErrorDescription2					:= ' ';	
	ELSIF NOT fbVirtualAxis.pSetPos.Error AND eState = E_Station.eResetting AND arrFbAllarm[23].bActive THEN
			arrFbAllarm[23].Clear(nTimeStamp := 0, bResetConfirmation := FALSE);
	END_IF;
	
	IF fbCamTableSelectAxisZ.Error AND NOT arrFbAllarm[24].bActive THEN
		arrFbAllarm[24].ipArguments.Clear().AddUDInt(fbCamTableSelectAxisZ.ErrorID);		
		arrFbAllarm[24].Raise(nTimeStamp := 0);		
    	udiErrorID							:= 1154;
    	udiErrorID							:= udiErrorID + iStationIndex;
    	sErrorDescription					:= CONCAT('Błąd generowania krzywki osi Z, MC_CamTableSelect.ErrorID:', UDINT_TO_STRING(fbCamTableSelectAxisZ.ErrorID));
    	sErrorDescription2					:= ' ';	
	ELSIF NOT fbCamTableSelectAxisZ.Error AND eState = E_Station.eResetting AND arrFbAllarm[24].bActive THEN
			arrFbAllarm[24].Clear(nTimeStamp := 0, bResetConfirmation := FALSE);
	END_IF;
	
	IF fbCamTableSelectCatcher.Error AND NOT arrFbAllarm[25].bActive THEN
		arrFbAllarm[25].ipArguments.Clear().AddUDInt(fbCamTableSelectCatcher.ErrorID);		
		arrFbAllarm[25].Raise(nTimeStamp := 0);		
    	udiErrorID							:= 1155;
    	udiErrorID							:= udiErrorID + iStationIndex;
    	sErrorDescription					:= CONCAT('Błąd generowania krzywki osi prowadzenia słomki, MC_CamTableSelect.ErrorID:', UDINT_TO_STRING(fbCamTableSelectCatcher.ErrorID));
    	sErrorDescription2					:= ' ';	
	ELSIF NOT fbCamTableSelectCatcher.Error AND eState = E_Station.eResetting AND arrFbAllarm[25].bActive THEN
			arrFbAllarm[25].Clear(nTimeStamp := 0, bResetConfirmation := FALSE);
	END_IF;
	
	IF fbCamInAxisZ.Error AND NOT arrFbAllarm[26].bActive THEN
		arrFbAllarm[26].ipArguments.Clear().AddUDInt(fbCamInAxisZ.ErrorID);		
		arrFbAllarm[26].Raise(nTimeStamp := 0);		
    	udiErrorID							:= 1156;
    	udiErrorID							:= udiErrorID + iStationIndex;
    	sErrorDescription					:= CONCAT('Błąd synchronizacji osi Z, MC_CamIn.ErrorID: ', UDINT_TO_STRING(fbCamInAxisZ.ErrorID));
    	sErrorDescription2					:= ' ';	
	ELSIF NOT fbCamInAxisZ.Error AND eState = E_Station.eResetting AND arrFbAllarm[26].bActive THEN
			arrFbAllarm[26].Clear(nTimeStamp := 0, bResetConfirmation := FALSE);
	END_IF;
	
	IF fbCamInAxisCatcher.Error AND NOT arrFbAllarm[27].bActive THEN
		arrFbAllarm[27].ipArguments.Clear().AddUDInt(fbCamInAxisCatcher.ErrorID);		
		arrFbAllarm[27].Raise(nTimeStamp := 0);		
    	udiErrorID							:= 1157;
    	udiErrorID							:= udiErrorID + iStationIndex;
    	sErrorDescription					:= CONCAT('Błąd synchronizacji osi prowadzenia słomki, MC_CamIn.ErrorID:', UDINT_TO_STRING(fbCamInAxisCatcher.ErrorID));
    	sErrorDescription2					:= ' ';	
	ELSIF NOT fbCamInAxisCatcher.Error AND eState = E_Station.eResetting AND arrFbAllarm[27].bActive THEN
			arrFbAllarm[27].Clear(nTimeStamp := 0, bResetConfirmation := FALSE);
	END_IF;
	
	IF fbCamOutAxisZ.Error AND NOT arrFbAllarm[28].bActive THEN
		arrFbAllarm[28].ipArguments.Clear().AddUDInt(fbCamOutAxisZ.ErrorID);		
		arrFbAllarm[28].Raise(nTimeStamp := 0);		
    	udiErrorID							:= 1158;
    	udiErrorID							:= udiErrorID + iStationIndex;
    	sErrorDescription					:= CONCAT('Błąd rozsynchronizacji osi Z, MCCamOut.ErrorID:', UDINT_TO_STRING(fbCamOutAxisZ.ErrorID));
    	sErrorDescription2					:= ' ';	
	ELSIF NOT fbCamOutAxisZ.Error AND eState = E_Station.eResetting AND arrFbAllarm[28].bActive THEN
			arrFbAllarm[28].Clear(nTimeStamp := 0, bResetConfirmation := FALSE);
	END_IF;
	
	IF fbCamOutAxisCatcher.Error AND NOT arrFbAllarm[29].bActive THEN
		arrFbAllarm[29].ipArguments.Clear().AddUDInt(fbCamOutAxisCatcher.ErrorID);		
		arrFbAllarm[29].Raise(nTimeStamp := 0);		
    	udiErrorID							:= 1159;
    	udiErrorID							:= udiErrorID + iStationIndex;
    	sErrorDescription					:= CONCAT('Błąd rozsynchronizacji osi prowadzenia słomki, MCCamOut.ErrorID:', UDINT_TO_STRING(fbCamOutAxisCatcher.ErrorID));
    	sErrorDescription2					:= ' ';	
	ELSIF NOT fbCamOutAxisCatcher.Error AND eState = E_Station.eResetting AND arrFbAllarm[29].bActive THEN
			arrFbAllarm[29].Clear(nTimeStamp := 0, bResetConfirmation := FALSE);
	END_IF;
	
	FOR i:= 0 TO 23 DO
		bError S= arrFbAllarm[i].bActive;
	END_FOR
	
ELSE
	bError := FALSE;
END_IF


//******************PRZEJŚCIE DO eERROR*****************************


IF bError AND NOT bStateError THEN
	IF eLastState = E_Station.eRunning THEN
		bCycleNotDone 			:= FALSE;
	END_IF
	eState := E_Station.eError;
	ResetCommands();
END_IF

//****************WYŚWIETLANIE STATUSU BLEDU***********************

(*Wyświetlanie błedu na wyjściu*)
bError;

(*Przepisywanie nazwy stacji*)
sErrorStationName := wsLiteral_TO_UTF8(wsStationName);

(*Kasowanie casów resettingu*)
//IF  udiErrorID-iStationIndex <>3 THEN
//	iErrorResseting3	:=	0;
//END_IF
END_ACTION

ACTION FBs:
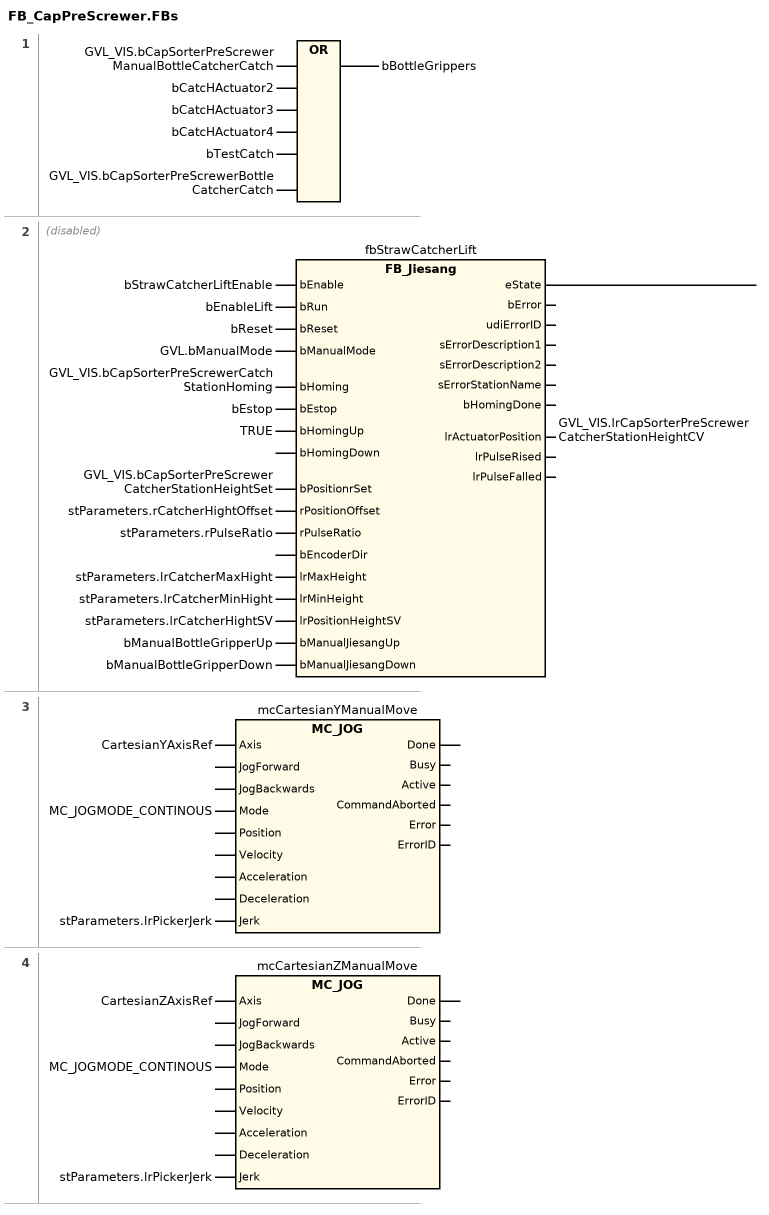
// NETWORK 1
bBottleGrippers := GVL_VIS.bCapSorterPreScrewerManualBottleCatcherCatch OR bCatcHActuator2 OR bCatcHActuator3 OR bCatcHActuator4 OR bTestCatch OR GVL_VIS.bCapSorterPreScrewerBottleCatcherCatch;

// NETWORK 2 (disabled)
// fbStrawCatcherLift(
//     bEnable := bStrawCatcherLiftEnable,
//     bRun := bEnableLift,
//     bReset := bReset,
//     bManualMode := GVL.bManualMode,
//     bHoming := GVL_VIS.bCapSorterPreScrewerCatchStationHoming,
//     bEstop := bEstop,
//     bHomingUp := TRUE,
//     bPositionrSet := GVL_VIS.bCapSorterPreScrewerCatcherStationHeightSet,
//     rPositionOffset := stParameters.rCatcherHightOffset,
//     rPulseRatio := stParameters.rPulseRatio,
//     lrMaxHeight := stParameters.lrCatcherMaxHight,
//     lrMinHeight := stParameters.lrCatcherMinHight,
//     lrPositionHeightSV := stParameters.lrCatcherHightSV,
//     bManualJiesangUp := bManualBottleGripperUp,
//     bManualJiesangDown := bManualBottleGripperDown,
//     lrActuatorPosition => GVL_VIS.lrCapSorterPreScrewerCatcherStationHeightCV); // FB_Jiesang

// NETWORK 3
mcCartesianYManualMove(
    Axis := CartesianYAxisRef,
    Mode := MC_JOGMODE_CONTINOUS,
    Jerk := stParameters.lrPickerJerk); // MC_JOG

// NETWORK 4
mcCartesianZManualMove(
    Axis := CartesianZAxisRef,
    Mode := MC_JOGMODE_CONTINOUS,
    Jerk := stParameters.lrPickerJerk); // MC_JOG

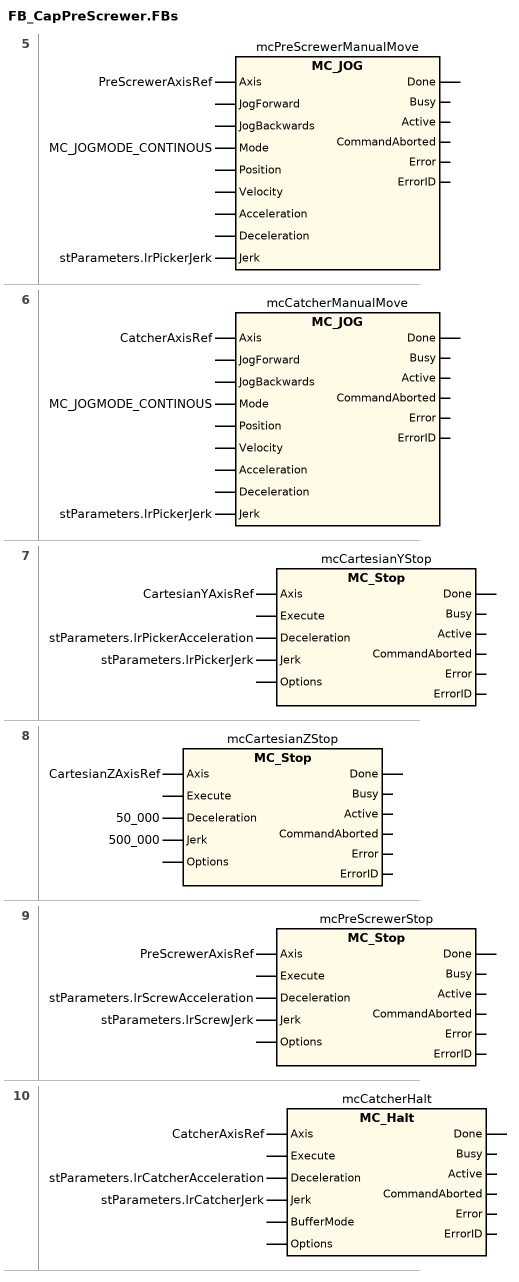
// NETWORK 5
mcPreScrewerManualMove(
    Axis := PreScrewerAxisRef,
    Mode := MC_JOGMODE_CONTINOUS,
    Jerk := stParameters.lrPickerJerk); // MC_JOG

// NETWORK 6
mcCatcherManualMove(Axis := CatcherAxisRef, Mode := MC_JOGMODE_CONTINOUS, Jerk := stParameters.lrPickerJerk); // MC_JOG

// NETWORK 7
mcCartesianYStop(
    Axis := CartesianYAxisRef,
    Deceleration := stParameters.lrPickerAcceleration,
    Jerk := stParameters.lrPickerJerk); // MC_Stop

// NETWORK 8
mcCartesianZStop(Axis := CartesianZAxisRef, Deceleration := 50_000, Jerk := 500_000); // MC_Stop

// NETWORK 9
mcPreScrewerStop(
    Axis := PreScrewerAxisRef,
    Deceleration := stParameters.lrScrewAcceleration,
    Jerk := stParameters.lrScrewJerk); // MC_Stop

// NETWORK 10
mcCatcherHalt(
    Axis := CatcherAxisRef,
    Deceleration := stParameters.lrCatcherAcceleration,
    Jerk := stParameters.lrCatcherJerk); // MC_Halt

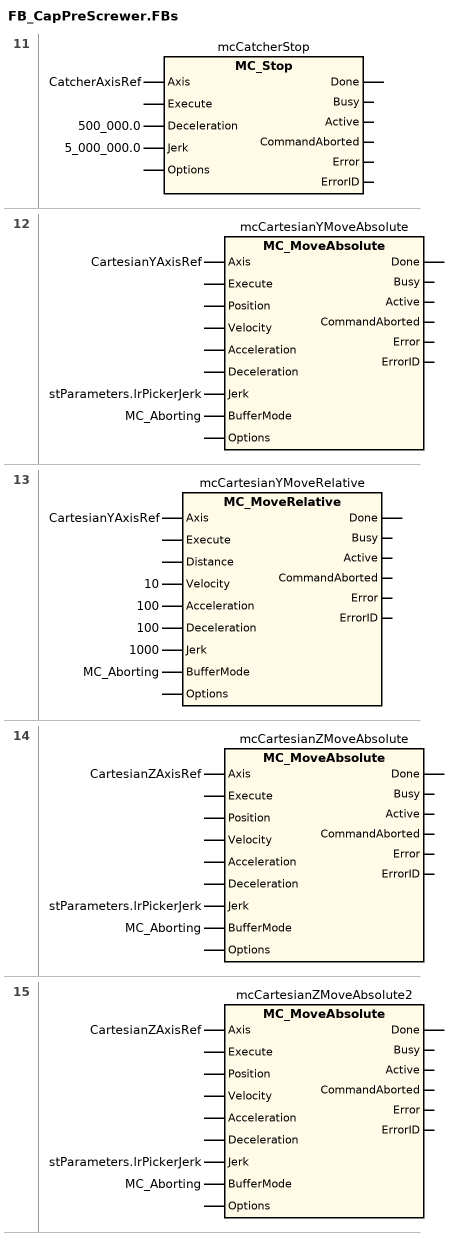
// NETWORK 11
mcCatcherStop(Axis := CatcherAxisRef, Deceleration := 500_000.0, Jerk := 5_000_000.0); // MC_Stop

// NETWORK 12
mcCartesianYMoveAbsolute(
    Axis := CartesianYAxisRef,
    Jerk := stParameters.lrPickerJerk,
    BufferMode := MC_Aborting); // MC_MoveAbsolute

// NETWORK 13
mcCartesianYMoveRelative(
    Axis := CartesianYAxisRef,
    Velocity := 10,
    Acceleration := 100,
    Deceleration := 100,
    Jerk := 1000,
    BufferMode := MC_Aborting); // MC_MoveRelative

// NETWORK 14
mcCartesianZMoveAbsolute(
    Axis := CartesianZAxisRef,
    Jerk := stParameters.lrPickerJerk,
    BufferMode := MC_Aborting); // MC_MoveAbsolute

// NETWORK 15
mcCartesianZMoveAbsolute2(
    Axis := CartesianZAxisRef,
    Jerk := stParameters.lrPickerJerk,
    BufferMode := MC_Aborting); // MC_MoveAbsolute

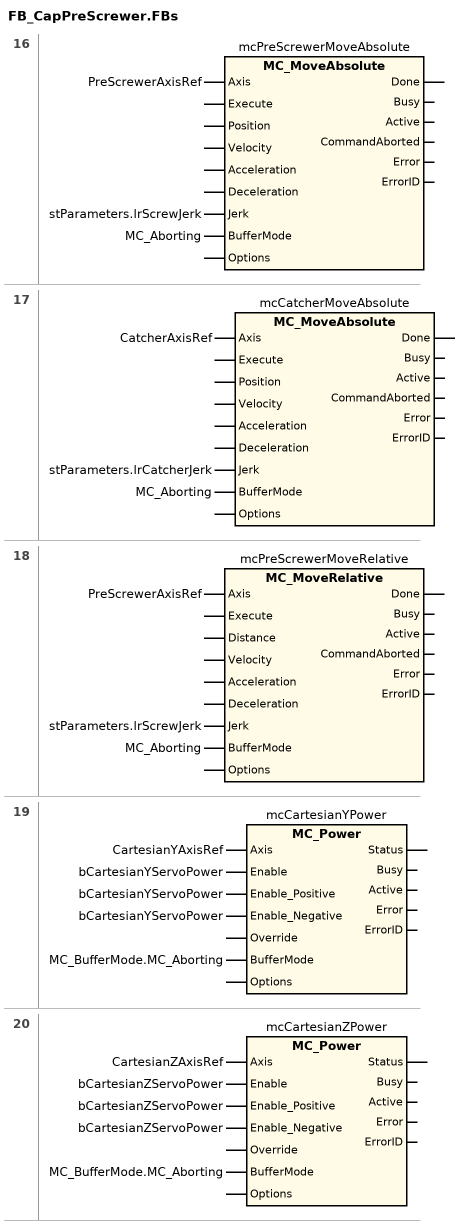
// NETWORK 16
mcPreScrewerMoveAbsolute(
    Axis := PreScrewerAxisRef,
    Jerk := stParameters.lrScrewJerk,
    BufferMode := MC_Aborting); // MC_MoveAbsolute

// NETWORK 17
mcCatcherMoveAbsolute(Axis := CatcherAxisRef, Jerk := stParameters.lrCatcherJerk, BufferMode := MC_Aborting); // MC_MoveAbsolute

// NETWORK 18
mcPreScrewerMoveRelative(
    Axis := PreScrewerAxisRef,
    Jerk := stParameters.lrScrewJerk,
    BufferMode := MC_Aborting); // MC_MoveRelative

// NETWORK 19
mcCartesianYPower(
    Axis := CartesianYAxisRef,
    Enable := bCartesianYServoPower,
    Enable_Positive := bCartesianYServoPower,
    Enable_Negative := bCartesianYServoPower,
    BufferMode := MC_BufferMode.MC_Aborting); // MC_Power

// NETWORK 20
mcCartesianZPower(
    Axis := CartesianZAxisRef,
    Enable := bCartesianZServoPower,
    Enable_Positive := bCartesianZServoPower,
    Enable_Negative := bCartesianZServoPower,
    BufferMode := MC_BufferMode.MC_Aborting); // MC_Power

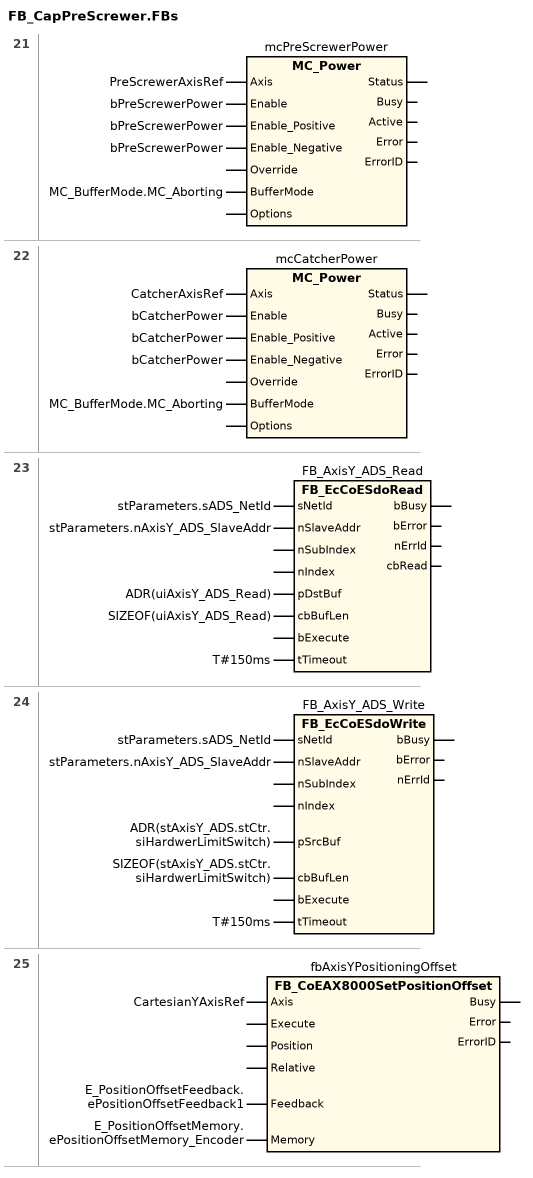
// NETWORK 21
mcPreScrewerPower(
    Axis := PreScrewerAxisRef,
    Enable := bPreScrewerPower,
    Enable_Positive := bPreScrewerPower,
    Enable_Negative := bPreScrewerPower,
    BufferMode := MC_BufferMode.MC_Aborting); // MC_Power

// NETWORK 22
mcCatcherPower(
    Axis := CatcherAxisRef,
    Enable := bCatcherPower,
    Enable_Positive := bCatcherPower,
    Enable_Negative := bCatcherPower,
    BufferMode := MC_BufferMode.MC_Aborting); // MC_Power

// NETWORK 23
FB_AxisY_ADS_Read(
    sNetId := stParameters.sADS_NetId,
    nSlaveAddr := stParameters.nAxisY_ADS_SlaveAddr,
    pDstBuf := ADR(uiAxisY_ADS_Read),
    cbBufLen := SIZEOF(uiAxisY_ADS_Read),
    tTimeout := T#150ms); // FB_EcCoESdoRead

// NETWORK 24
FB_AxisY_ADS_Write(
    sNetId := stParameters.sADS_NetId,
    nSlaveAddr := stParameters.nAxisY_ADS_SlaveAddr,
    pSrcBuf := ADR(stAxisY_ADS.stCtr.siHardwerLimitSwitch),
    cbBufLen := SIZEOF(stAxisY_ADS.stCtr.siHardwerLimitSwitch),
    tTimeout := T#150ms); // FB_EcCoESdoWrite

// NETWORK 25
fbAxisYPositioningOffset(
    Axis := CartesianYAxisRef,
    Feedback := E_PositionOffsetFeedback.ePositionOffsetFeedback1,
    Memory := E_PositionOffsetMemory.ePositionOffsetMemory_Encoder); // FB_CoEAX8000SetPositionOffset

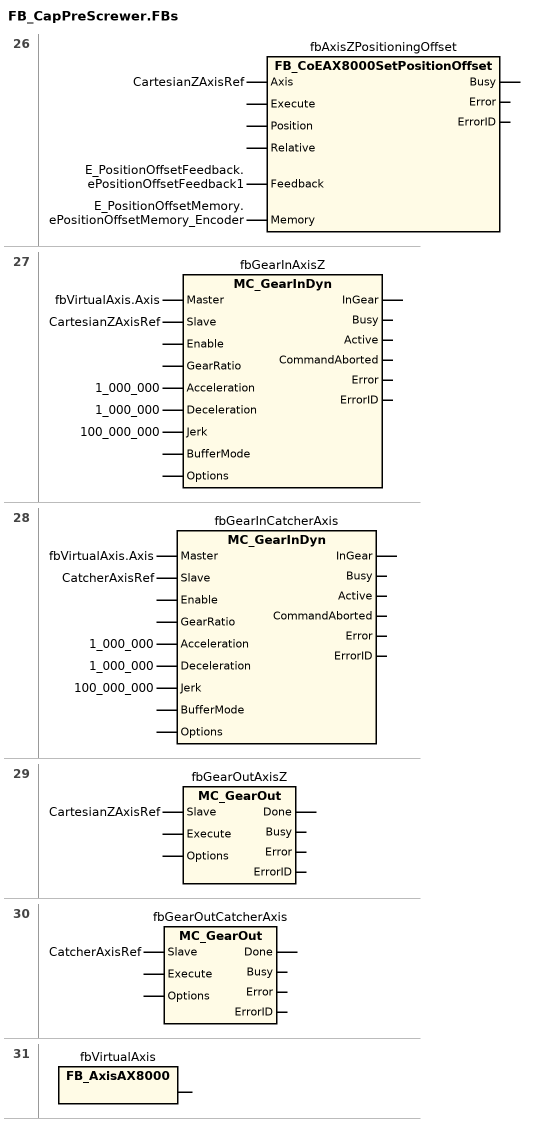
// NETWORK 26
fbAxisZPositioningOffset(
    Axis := CartesianZAxisRef,
    Feedback := E_PositionOffsetFeedback.ePositionOffsetFeedback1,
    Memory := E_PositionOffsetMemory.ePositionOffsetMemory_Encoder); // FB_CoEAX8000SetPositionOffset

// NETWORK 27
fbGearInAxisZ(
    Master := fbVirtualAxis.Axis,
    Slave := CartesianZAxisRef,
    Acceleration := 1_000_000,
    Deceleration := 1_000_000,
    Jerk := 100_000_000); // MC_GearInDyn

// NETWORK 28
fbGearInCatcherAxis(
    Master := fbVirtualAxis.Axis,
    Slave := CatcherAxisRef,
    Acceleration := 1_000_000,
    Deceleration := 1_000_000,
    Jerk := 100_000_000); // MC_GearInDyn

// NETWORK 29
fbGearOutAxisZ(Slave := CartesianZAxisRef); // MC_GearOut

// NETWORK 30
fbGearOutCatcherAxis(Slave := CatcherAxisRef); // MC_GearOut

// NETWORK 31
fbVirtualAxis(); // FB_AxisAX8000

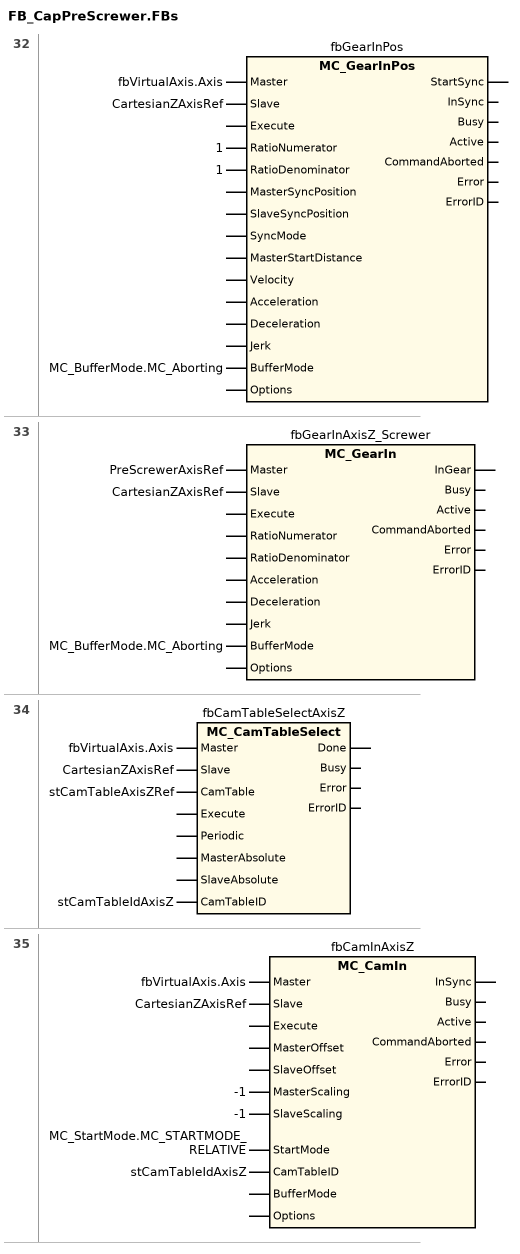
// NETWORK 32
fbGearInPos(
    Master := fbVirtualAxis.Axis,
    Slave := CartesianZAxisRef,
    RatioNumerator := 1,
    RatioDenominator := 1,
    BufferMode := MC_BufferMode.MC_Aborting); // MC_GearInPos

// NETWORK 33
fbGearInAxisZ_Screwer(
    Master := PreScrewerAxisRef,
    Slave := CartesianZAxisRef,
    BufferMode := MC_BufferMode.MC_Aborting); // MC_GearIn

// NETWORK 34
fbCamTableSelectAxisZ(
    Master := fbVirtualAxis.Axis,
    Slave := CartesianZAxisRef,
    CamTable := stCamTableAxisZRef,
    CamTableID := stCamTableIdAxisZ); // MC_CamTableSelect

// NETWORK 35
fbCamInAxisZ(
    Master := fbVirtualAxis.Axis,
    Slave := CartesianZAxisRef,
    MasterScaling := -1,
    SlaveScaling := -1,
    StartMode := MC_StartMode.MC_STARTMODE_RELATIVE,
    CamTableID := stCamTableIdAxisZ); // MC_CamIn

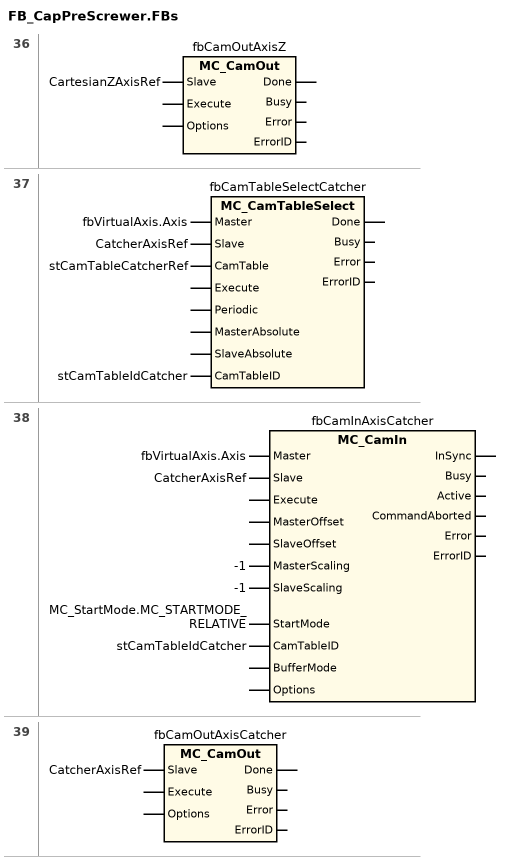
// NETWORK 36
fbCamOutAxisZ(Slave := CartesianZAxisRef); // MC_CamOut

// NETWORK 37
fbCamTableSelectCatcher(
    Master := fbVirtualAxis.Axis,
    Slave := CatcherAxisRef,
    CamTable := stCamTableCatcherRef,
    CamTableID := stCamTableIdCatcher); // MC_CamTableSelect

// NETWORK 38
fbCamInAxisCatcher(
    Master := fbVirtualAxis.Axis,
    Slave := CatcherAxisRef,
    MasterScaling := -1,
    SlaveScaling := -1,
    StartMode := MC_StartMode.MC_STARTMODE_RELATIVE,
    CamTableID := stCamTableIdCatcher); // MC_CamIn

// NETWORK 39
fbCamOutAxisCatcher(Slave := CatcherAxisRef); // MC_CamOut
END_ACTION

ACTION Homing:
tonAxisYLagDetction(PT := T#250MS);

IF mcCartesianZPower.Status AND mcPreScrewerPower.Status AND mcCatcherPower.Status THEN
		
	IF bHoming THEN // Bazowanie - podjazd do góry i ustawienie obrotu
		IF NOT bAdvancedHoming THEN
			CASE iHomingCase OF
			
				0:
					mcCartesianYPower.Override			:=	100;			
					mcCartesianZPower.Override			:=	100;			
					mcPreScrewerPower.Override			:=	100;			
					mcCatcherPower.Override				:=	100;	
					                                    
					bCartesianYServoPower				:= TRUE;
					bCartesianZServoPower				:= TRUE;
					bPreScrewerPower					:= TRUE;
					bCatcherPower						:= TRUE;	
					                                    
					mcCartesianYManualMove.JogBackwards	:=FALSE;
					mcCartesianZManualMove.JogBackwards	:=FALSE;
					mcPreScrewerManualMove.JogBackwards	:=FALSE;
					mcCatcherManualMove.JogBackwards	:=FALSE;
					                                    
					mcCartesianYManualMove.JogForward	:=FALSE;
					mcCartesianZManualMove.JogForward	:=FALSE;
					mcPreScrewerManualMove.JogForward	:=FALSE;
					mcCatcherManualMove.JogForward		:=FALSE;
					bCycleNotDone						:= FALSE;				
					
					IF bAnyCapPresence THEN
						iHomingCase						:= iHomingCase	+	100;
					ELSE
						iHomingCase						:= iHomingCase	+	10;	
					END_IF
					
					bHomingDone							:= FALSE;
				
				10: 
        	
					//Otwórz chwytaki
					bCapCatcher1				:= FALSE;
					bCapCatcher2				:= FALSE;
					bCapCatcher3				:= FALSE;
					bCapCatcher4				:= FALSE;
					//Wyłącz ssawki
					bCapSucker[1]					:= FALSE;
					bCapSucker[2]					:= FALSE;
					bCapSucker[3]					:= FALSE;
					bCapSucker[4]					:= FALSE;
					//Otwórz chwytaki słomek
					bStrawCatchersOpen			:= TRUE;
					bStrawCatchersClose			:= FALSE;
					//Cofnij chwytaki słomek
					bStrawCatcherActuatorIn		:= TRUE;
					bStrawCatcherActuatorOut	:= FALSE;
					//Podjedź robotem i chwytakiem słomek w górę jak cofnięty chwytak słomek - bazuj podnośnik Jisang
					IF tonStrawCatcherIn.Q THEN	
						mcCartesianZMoveAbsolute.Execute		:= TRUE;		
						mcCartesianZMoveAbsolute.Position		:= 420;//stParameters.lrTopZPosition;
						mcCartesianZMoveAbsolute.Acceleration	:= stParameters.lrPickerAcceleration;
						mcCartesianZMoveAbsolute.Deceleration	:= stParameters.lrPickerAcceleration;
						mcCartesianZMoveAbsolute.Velocity		:= 200;//stParameters.lrPickerSpeed;			
						
						fbStrawCatcherLift.bHoming;//				:= TRUE;
						//fbStrawCatcherLift.bHomingUp;//			:= TRUE;
						GVL_VIS.bCapSorterPreScrewerCatchStationHoming			:= NOT fbStrawCatcherLift.bHomingDone;
						GVL_VIS.bCapSorterPreScrewerCatcherStationHeightSet		:= NOT GVL_VIS.bCapSorterPreScrewerCatchStationHoming AND NOT bStrawCatcherLiftInHomePos;
						bEnableLift												:= TRUE;
						//Następny krok
						iHomingCase								:= iHomingCase + 10;
					END_IF
					//Reset komendy ruchu osi X
					mcCartesianYMoveAbsolute.Execute		:= FALSE;
					
			
				20:		
					(*Czekam na pozycję Z w górze i ruszam osią poziomą X na pozycję pobierania i czekam na obie pozycje*)
					bHomingWithoutJiesang						:= FALSE;
	    	
					IF (CartesianZAxisRef.NcToPlc.ActPos > stParameters.lrTopZPosition - stParameters.lrBendingDistance) OR
						mcCartesianZMoveAbsolute.Done THEN
						
						mcCatcherMoveAbsolute.Execute			:= TRUE;		
						mcCatcherMoveAbsolute.Position			:= stParameters.lrCatcherCatchingPosition;
						mcCatcherMoveAbsolute.Acceleration		:= stParameters.lrCatcherAcceleration;
						mcCatcherMoveAbsolute.Deceleration		:= stParameters.lrCatcherAcceleration;
						mcCatcherMoveAbsolute.Velocity			:= 30;//stParameters.lrCatcherSpeed;
						
						//Jedź osią poziomą Y na pozycję pick
						mcCartesianYMoveAbsolute.Execute		:= TRUE;
						mcCartesianYMoveAbsolute.Position		:= stParameters.lrPickYPosition;
						mcCartesianYMoveAbsolute.Acceleration	:= stParameters.lrPickerAcceleration;
						mcCartesianYMoveAbsolute.Deceleration	:= stParameters.lrPickerAcceleration;
						mcCartesianYMoveAbsolute.Velocity		:= 150;//stParameters.lrPickerSpeed;
						
						//Ustaw obracarkę w pozycji
						mcPreScrewerMoveRelative.Execute		:= TRUE;
						mcPreScrewerMoveRelative.Distance		:=  -1 * DINT_TO_LREAL(LREAL_TO_DINT(PreScrewerAxisRef.NcToPlc.SetPos) MOD 360);
						mcPreScrewerMoveRelative.Acceleration	:= stParameters.lrScrewAcceleration;
						mcPreScrewerMoveRelative.Deceleration	:= stParameters.lrScrewAcceleration;
						mcPreScrewerMoveRelative.Velocity		:= 180;//stParameters.lrScrewSpeed;
					END_IF
					IF mcPreScrewerMoveRelative.Done THEN
						mcPreScrewerMoveRelative.Execute		:= FALSE;
						mcPreScrewerHome(Axis := PreScrewerAxisRef, HomingMode := MC_Direct, Position := 0, Execute := TRUE);					
					END_IF
					//Jak obie pozycje osiągnięte to następny krok
					IF mcCartesianYMoveAbsolute.Done AND mcCartesianZMoveAbsolute.Done AND mcPreScrewerHome.Done AND bStrawCatcherLiftInHomePos THEN
						//Reset komendy ruchu osi
						bCapsBlowON								:= TRUE;
						bCapBlow1 								:= TRUE;
						bCapBlow2 								:= TRUE;
						bCapBlow3 								:= TRUE;
						bCapBlow4 								:= TRUE;
						mcCartesianYMoveAbsolute.Execute		:= FALSE;
						mcCartesianZMoveAbsolute.Execute		:= FALSE;
						mcPreScrewerHome.Execute				:= FALSE;
						//Reset homingu podnośnika Jisang
						fbStrawCatcherLift.bHoming;//				:= FALSE;
						GVL_VIS.bCapSorterPreScrewerCatchStationHoming			:= FALSE;
						GVL_VIS.bCapSorterPreScrewerCatcherStationHeightSet		:= FALSE;
					//	bEnableLift												:= FALSE;						
						
						
						//fbStrawCatcherLift.bHomingUp;//			:= FALSE;
						//Wysuń chwytaki słomek jesli to potrzebuje recepta
						bStrawCatcherActuatorIn					:= NOT stParameters.bStrawCatcherON;
						bStrawCatcherActuatorOut				:= stParameters.bStrawCatcherON;
						//Następny krok
						iHomingCase								:= iHomingCase + 10;
					END_IF
				
				30:	//Koniec
				IF NOT bCapBlow1 AND NOT bCapBlow2 AND NOT bCapBlow3 AND NOT bCapBlow4 THEN
						eState								:= E_Station.eHomingDone;
						bHomingDone							:= TRUE;
						iHomingCase							:= 0; 
				END_IF
				
				
				
				
				
				100://Odrzut nasadek
						//Otwórz chwytaki gdy nakrętka była zakręcana
					bCapCatcher1				R= bCapScrewed;
					bCapCatcher2				R= bCapScrewed;
					bCapCatcher3				R= bCapScrewed;
					bCapCatcher4				R= bCapScrewed;

						//Otwórz chwytaki słomek
					bStrawCatchersOpen			:= TRUE;
					bStrawCatchersClose			:= FALSE;
						//Cofnij chwytaki słomek
					bStrawCatcherActuatorIn		:= TRUE;
					bStrawCatcherActuatorOut	:= FALSE;
										//Podjedź robotem i chwytakiem słomek w górę jak cofnięty chwytak słomek - bazuj podnośnik Jisang
					IF tonStrawCatcherIn.Q THEN	
						mcCartesianZMoveAbsolute.Execute		:= TRUE;		
						mcCartesianZMoveAbsolute.Position		:= 420;//stParameters.lrTopZPosition;
						mcCartesianZMoveAbsolute.Acceleration	:= stParameters.lrPickerAcceleration;
						mcCartesianZMoveAbsolute.Deceleration	:= stParameters.lrPickerAcceleration;
						mcCartesianZMoveAbsolute.Velocity		:= 200;//stParameters.lrPickerSpeed;	70		
	
						//Następny krok
						iHomingCase								:= iHomingCase + 10;
					END_IF
					//Reset komendy ruchu osi X
					mcCartesianYMoveAbsolute.Execute		:= FALSE;
					
				110:
									(*Czekam na pozycję Z w górze i ruszam osią poziomą X na pozycję pobierania i czekam na obie pozycje*)
	    	
					IF (CartesianZAxisRef.NcToPlc.ActPos > stParameters.lrTopZPosition - stParameters.lrBendingDistance) OR
						mcCartesianZMoveAbsolute.Done THEN
						
						mcCatcherMoveAbsolute.Execute			:= TRUE;		
						mcCatcherMoveAbsolute.Position			:= stParameters.lrCatcherCatchingPosition;
						mcCatcherMoveAbsolute.Acceleration		:= stParameters.lrCatcherAcceleration;
						mcCatcherMoveAbsolute.Deceleration		:= stParameters.lrCatcherAcceleration;
						mcCatcherMoveAbsolute.Velocity			:= 200;//stParameters.lrCatcherSpeed;	70
						
						//Jedź osią poziomą Y na pozycję pick
						mcCartesianYMoveAbsolute.Execute		:= TRUE;
						mcCartesianYMoveAbsolute.Position		:= 3.0;
						mcCartesianYMoveAbsolute.Acceleration	:= stParameters.lrPickerAcceleration;
						mcCartesianYMoveAbsolute.Deceleration	:= stParameters.lrPickerAcceleration;
						mcCartesianYMoveAbsolute.Velocity		:= 200;//stParameters.lrPickerSpeed;	20
						
					END_IF
					
					//Jak obie pozycje osiągnięte to następny krok
					IF mcCartesianYMoveAbsolute.Done AND mcCartesianZMoveAbsolute.Done AND mcPreScrewerHome.Done AND fbStrawCatcherLift.bHomingDone THEN
						//Reset komendy ruchu osi

						mcCartesianYMoveAbsolute.Execute						:= FALSE;
						mcCartesianZMoveAbsolute.Execute						:= FALSE;
						mcPreScrewerHome.Execute								:= FALSE;
						//Reset homingu podnośnika Jisang
						fbStrawCatcherLift.bHoming;//				:= FALSE;
						GVL_VIS.bCapSorterPreScrewerCatchStationHoming			:= FALSE;
						GVL_VIS.bCapSorterPreScrewerCatcherStationHeightSet		:= FALSE;
						bEnableLift												:= FALSE;						
						//fbStrawCatcherLift.bHomingUp;//			:= FALSE;
						//Następny krok
						iHomingCase								:= iHomingCase + 10;
					END_IF		
					
					120:
					mcCartesianZMoveAbsolute.Execute			:= TRUE;		
					mcCartesianZMoveAbsolute.Position			:= 400;//stParameters.lrTopZPosition;
					mcCartesianZMoveAbsolute.Acceleration		:= stParameters.lrPickerAcceleration;
					mcCartesianZMoveAbsolute.Deceleration		:= stParameters.lrPickerAcceleration;
					mcCartesianZMoveAbsolute.Velocity			:= 200;//stParameters.lrPickerSpeed;	70
						
						IF mcCartesianZMoveAbsolute.Done THEN
							mcCartesianZMoveAbsolute.Execute	:= FALSE;	
								//Otwórz chwytaki
							bCapCatcher1						:= FALSE;
							bCapCatcher2						:= FALSE;
							bCapCatcher3						:= FALSE;
							bCapCatcher4						:= FALSE;
								//Wyłącz ssawki         		
							bCapSucker[1]							:= FALSE;
							bCapSucker[2]							:= FALSE;
							bCapSucker[3]							:= FALSE;
							bCapSucker[4]							:= FALSE;
							bCapsBlowON							:= TRUE;
							bCapBlow1 							:= TRUE;
							bCapBlow2 							:= TRUE;
							bCapBlow3 							:= TRUE;
							bCapBlow4 							:= TRUE;
							iHomingCase							:= iHomingCase + 10;
						END_IF
						
					130:
					IF NOT bCapBlow1 AND NOT bCapBlow2 AND NOT bCapBlow3 AND NOT bCapBlow4 THEN
						iHomingCase							:= 10; 
					END_IF
				
				
				
			END_CASE
		ELSE
			CASE iHomingCase OF
				0:
				mcCartesianYPower.Override					:=	100;			
				mcCartesianZPower.Override					:=	100;			
				mcPreScrewerPower.Override					:=	100;			
				mcCatcherPower.Override						:=	100;
				                                    		
				bCartesianYServoPower						:= TRUE;
				bCartesianZServoPower						:= TRUE;
				bPreScrewerPower							:= TRUE;
				bCatcherPower								:= TRUE;	
				                                    		
				mcCartesianYManualMove.JogBackwards			:=FALSE;
				mcCartesianZManualMove.JogBackwards			:=FALSE;
				mcPreScrewerManualMove.JogBackwards			:=FALSE;
				mcCatcherManualMove.JogBackwards			:=FALSE;
				                                    		
				mcCartesianYManualMove.JogForward			:=FALSE;
				mcCartesianZManualMove.JogForward			:=FALSE;
				mcPreScrewerManualMove.JogForward			:=FALSE;
				mcCatcherManualMove.JogForward				:=FALSE;
				bCycleNotDone								:= FALSE;
				iHomingCase									:= 10;
				bHomingDone									:= FALSE;
				
				10:
					//Otwórz chwytaki
				bCapCatcher1										:= FALSE;
				bCapCatcher2										:= FALSE;
				bCapCatcher3										:= FALSE;
				bCapCatcher4										:= FALSE;
				//Wyłącz ssawki             						
				bCapSucker[1]											:= FALSE;
				bCapSucker[2]											:= FALSE;
				bCapSucker[3]											:= FALSE;
				bCapSucker[4]											:= FALSE;
				//Otwórz chwytaki słomek    						
				bStrawCatchersOpen									:= TRUE;
				bStrawCatchersClose									:= FALSE;
				//Cofnij chwytaki słomek    						
				bStrawCatcherActuatorIn								:= TRUE;
				bStrawCatcherActuatorOut							:= FALSE;
				
					//Podjedź robotem i chwytakiem słomek w górę jak cofnięty chwytak słomek - bazuj podnośnik Jisang
					IF tonStrawCatcherIn.Q THEN	
						mcCartesianZMoveAbsolute.Execute				:= TRUE;		
						mcCartesianZMoveAbsolute.Position				:= 420;
						mcCartesianZMoveAbsolute.Acceleration			:= stParameters.lrPickerAcceleration;
						mcCartesianZMoveAbsolute.Deceleration			:= stParameters.lrPickerAcceleration;
						mcCartesianZMoveAbsolute.Velocity				:= 30;					                                     
						                                        		
						fbStrawCatcherLift.bHoming;//					:= TRUE;
						//fbStrawCatcherLift.bHomingUp;//					:= TRUE;
						GVL_VIS.bCapSorterPreScrewerCatchStationHoming			:= NOT fbStrawCatcherLift.bHomingDone;
						GVL_VIS.bCapSorterPreScrewerCatcherStationHeightSet		:= NOT GVL_VIS.bCapSorterPreScrewerCatchStationHoming AND NOT bStrawCatcherLiftInHomePos;
						bEnableLift												:= TRUE;
						//Następny krok
						iHomingCase										:= iHomingCase + 10;
					END_IF
				//Reset komendy ruchu osi X
				mcCartesianYMoveAbsolute.Execute					:= FALSE;
				
				20:
	(*Czekam na pozycję Z w górze i ruszam osią poziomą X na pozycję pobierania i czekam na obie pozycje*)
				bHomingWithoutJiesang						:= FALSE;
	
					IF (CartesianZAxisRef.NcToPlc.ActPos > stParameters.lrTopZPosition - stParameters.lrBendingDistance) OR
						mcCartesianZMoveAbsolute.Done THEN
						
						mcCatcherMoveAbsolute.Execute				:= TRUE;		
						mcCatcherMoveAbsolute.Position				:= stParameters.lrCatcherCatchingPosition;
						mcCatcherMoveAbsolute.Acceleration			:= stParameters.lrCatcherAcceleration;
						mcCatcherMoveAbsolute.Deceleration			:= stParameters.lrCatcherAcceleration;
						mcCatcherMoveAbsolute.Velocity				:= 30;
						                                            
							//Ustaw obracarkę w pozycji             
						mcPreScrewerMoveRelative.Execute			:= TRUE;
						mcPreScrewerMoveRelative.Distance			:=  -1 * DINT_TO_LREAL(LREAL_TO_DINT(PreScrewerAxisRef.NcToPlc.SetPos) MOD 360);
						mcPreScrewerMoveRelative.Acceleration		:= stParameters.lrScrewAcceleration;
						mcPreScrewerMoveRelative.Deceleration		:= stParameters.lrScrewAcceleration;
						mcPreScrewerMoveRelative.Velocity			:= 180;//stParameters.lrScrewSpeed;	
					END_IF			

					IF mcPreScrewerMoveRelative.Done AND mcCartesianZMoveAbsolute.Done AND 	fbStrawCatcherLift.bHomingDone THEN
						tonAxisYLagDetction.IN						:= FALSE;
						mcPreScrewerMoveRelative.Execute			:= FALSE;
						mcCatcherMoveAbsolute.Execute				:= FALSE;
						mcCartesianZMoveAbsolute.Execute			:= FALSE;
						iHomingCase									:= iHomingCase + 10;
					END_IF
				
				30:
				//Ustawiamy moment osi Y na 15%
				stAxisY_ADS.stCtr.uiNegativeTorqueLimit				:= 500;
				stAxisY_ADS.stCtr.uiPositiveTorqueLimit				:= 500; 
				uiAxisYTorqueLimit									:= 500;	
				mcCartesianYManualMove.JogForward					:= FALSE;
				mcCartesianYManualMove.JogBackwards					:= TRUE;
				mcCartesianYManualMove.Velocity						:= 5; 
				iHomingCase											:= iHomingCase + 10;
				
				40://Detekcja lag'a 
				tonAxisYLagDetction.IN								:= (ABS(CartesianYAxisRef.NcToPlc.PosDiff) >= 5.0);

					IF tonAxisYLagDetction.Q THEN
						mcCartesianYManualMove.JogBackwards			:= FALSE;
						iHomingCase									:= iHomingCase + 10;
					END_IF	
				
				50:
				mcCartesianYMoveRelative.Distance					:= 20;
				mcCartesianYMoveRelative.Execute					:= TRUE;
				
					IF mcCartesianYMoveRelative.Done THEN
						mcCartesianYMoveRelative.Execute			:= FALSE;
						iHomingCase									:= iHomingCase + 10;
					END_IF
				
				60:
				bCartesianYServoPower								:= FALSE;
				fbAxisYPositioningOffset.Position					:= 0;
				
					IF CartesianYAxisRef.Status.Disabled THEN
						iHomingCase									:= iHomingCase + 10;
					END_IF
					
				70:
				fbAxisYPositioningOffset.Execute					:= TRUE;
				
					IF 	fbAxisYPositioningOffset.Busy THEN
						iHomingCase									:= iHomingCase + 10;
					END_IF
				
				80:
				IF NOT fbAxisYPositioningOffset.Busy THEN	
					fbAxisYPositioningOffset.Execute				:= FALSE;
					bCartesianYServoPower							:= TRUE;
					stAxisY_ADS.stCtr.uiNegativeTorqueLimit			:= 2000;	//200%
					stAxisY_ADS.stCtr.uiPositiveTorqueLimit			:= 2000;	//200%
					iHomingCase										:= iHomingCase + 10;
				END_IF
				
				90:	
				bCapsBlowON											:= TRUE;
				bCapBlow1 											:= TRUE;
				bCapBlow2 											:= TRUE;
				bCapBlow3 											:= TRUE;
                bCapBlow4 											:= TRUE;
				iHomingCase											:= iHomingCase + 10;
				
				100://Oddmuch
				IF NOT bCapBlow1 AND NOT bCapBlow2 AND NOT bCapBlow3 AND NOT bCapBlow4 THEN
					iHomingCase										:= iHomingCase + 10;
				END_IF	
				
				110://Jedź osią poziomą Y na pozycję pick					
				mcCartesianYMoveAbsolute.Execute					:= TRUE;
				mcCartesianYMoveAbsolute.Position					:= stParameters.lrPickYPosition;
				mcCartesianYMoveAbsolute.Acceleration				:= stParameters.lrPickerAcceleration;
				mcCartesianYMoveAbsolute.Deceleration				:= stParameters.lrPickerAcceleration;
				mcCartesianYMoveAbsolute.Velocity					:= 30;//stParameters.lrPickerSpeed;
				
					IF mcCartesianYMoveAbsolute.Done THEN	//Koniec
						mcCartesianYMoveAbsolute.Execute			:= FALSE;
						eState										:= E_Station.eHomingDone;
						bHomingDone									:= TRUE;
						iHomingCase									:= 0; 
					END_IF	
					
			END_CASE
		END_IF
	END_IF
END_IF
END_ACTION

ACTION ManualMovements:
tonVacuumWatchdog(PT	:= stParameters.tTimeVacuumWatchdog);
trStepButton(CLK 		:= bStepButton OR (stCommandsIn.bPendantRightwardMovement AND diManualModeCase<>0));
rtSetEncoderOffsetAxisZ(CLK := bSetEncoderOffsetAxisZ);

// Wyjście z trybu manualnego
	IF NOT bManualMovement THEN		
		ResetCommands();		
		eState											:= E_Station.eReady;
	END_IF
	
	IF mcCartesianYManualMove.Done OR mcCartesianZManualMove.Done OR mcPreScrewerManualMove.Done OR mcCatcherManualMove.Done THEN
		bHomingDone										:= FALSE;
	END_IF

	//Zmiana prędkości plotera na kasecie sterowniczej
		rtPendantRightLeftFast(CLK 	:= stCommandsIn.bPendantRightLeftFast);
		ftPendantRightLeftFast(CLK 	:= stCommandsIn.bPendantRightLeftFast);	
		bChangeSpeedRightLeft 		S= (rtPendantRightLeftFast.Q OR ftPendantRightLeftFast.Q);	
		bChangeSpeedRightLeft 		R= NOT CartesianYAxisRef.Status.Moving;
		
